(* CoDeSys 2.3.9.41 project: KS Griazovetskaya(ver27.07.20, manStopN0204).pro *)
(* Libraries: PID_Regulators.lib 6.11.19 15:29:27, Util.lib 18.5.10 15:14:28, STANDARD.LIB 4.10.05 11:14:46, IECSFC.LIB 13.4.06 15:51:28, ANALYZATION.LIB 5.10.99 09:05:06 *)

(* PLC configuration (modules and I/O channels)
Fast discrete inputs [I_SIMPLE_INPUT] node 0, in %IB0 out %QB0 {Filtrationtime = 10}
  DD1_DI0 AT %IX0.0 [BitInput] резерв
  DD1_DI1 AT %IX0.1 [BitInput] резерв
  DD1_DI2 AT %IX0.2 [BitInput] резерв
  DD1_DI3 AT %IX0.3 [BitInput] резерв
Discrete inputs [ID130] node 1, in %IB1 out %QB1 {Filtrationtime_GeneralINP = 10; Visibility = No; PinCount = 12}
  AT %IB1.0 [ByteInput] 8 discrete inputs
  AT %IB1.1 [ByteInput] 4 discrete inputs
Discrete outputs [ID131] node 2, in %IB2 out %QB2 {SafeValueByte = 0; SafeValueByteM = 0; Visibility = No; PinCount = 12}
  AT %QB2.0 [ByteOutput] 8 discrete outputs
  AT %QB2.1 [ByteOutput] 4 discrete outputs
Fast analog inputs [ID125] node 3, in %IB3 out %QB3 {Flt_Comm = 50Hz 2Por}
  DD1_AI0 AT %IR3.0 [FloatInputP] AI #1 - датчик температуры в помещении (метран) {AIN_TYPE = 4-20 mA; Peak_Filtr = 200; Flt_Ch = Off; TauRC = 10; MinFV = 0; MaxFV = 100}
  DD1_AI1 AT %IR3.1 [FloatInputP] AI #2 - расходомер FT01.01 (на входе, до отстойника) {AIN_TYPE = 4-20 mA; Peak_Filtr = 200; Flt_Ch = Off; TauRC = 10; MinFV = 0; MaxFV = 600}
  DD1_AI2 AT %IR3.2 [FloatInputP] AI #3 - расходомер FT01.02 (на выходе, после отстойника) {AIN_TYPE = 4-20 mA; Peak_Filtr = 200; Flt_Ch = Off; TauRC = 10; MinFV = 0; MaxFV = 600}
  DD1_AI3 AT %IR3.3 [FloatInputP] AI #4 - рН-метр QE01.01 (на входе, до отстойника) {AIN_TYPE = 4-20 mA; Peak_Filtr = 200; Flt_Ch = Off; TauRC = 10; MinFV = 0; MaxFV = 14}
  DD1_AI4 AT %IR3.4 [FloatInputP] AI #5 - рН-метр QE01.02 (на выходе, после отстойника) {AIN_TYPE = 4-20 mA; Peak_Filtr = 200; Flt_Ch = Off; TauRC = 10; MinFV = 0; MaxFV = 14}
  DD1_AI5 AT %IR3.5 [FloatInputP] AI #6 - сигнал от ФПК, давление на входе {AIN_TYPE = 4-20 mA; Peak_Filtr = 200; Flt_Ch = Off; TauRC = 10; MinFV = 0; MaxFV = 16}
  DD1_AI6 AT %IR3.6 [FloatInputP] AI #7 - резерв {AIN_TYPE = 4-20 mA; Peak_Filtr = 200; Flt_Ch = Off; TauRC = 10; MinFV = 0; MaxFV = 20000.0}
  DD1_AI7 AT %IR3.7 [FloatInputP] AI#8 - резерв {AIN_TYPE = 4-20 mA; Peak_Filtr = 200; Flt_Ch = Off; TauRC = 10; MinFV = 0; MaxFV = 20000.0}
  AT %IW3.8 [WordInput] AI read time (10ms)
Analog outputs [ID126] node 4, in %IB4 out %QB4
  DD1_AO0 AT %QR4.0 [FloatOutputP] AO #1 - управление ЧРП Н01.05 (поддержание расхода по расходомеру FT01.02) {AOUT_TYPE = 4-20 mA; SafeValueREAL = 0.0}
  DD1_AO1 AT %QR4.1 [FloatOutputP] AO #2 - управление ЧРП НД08.03/01 (подача флокулянта на входе, до отстойника, по FT01.01) {AOUT_TYPE = 4-20 mA; SafeValueREAL = 0.0}
  DD1_AO2 AT %QR4.2 [FloatOutputP] AO #3 - управление ЧРП НД08.03/02 (подача флокулянта на входе, до отстойника, по FT01.01) {AOUT_TYPE = 4-20 mA; SafeValueREAL = 0.0}
  DD1_AO3 AT %QR4.3 [FloatOutputP] AO #4 - управление НД05.02/01 (подача 10%NaCl из УПГ на входе, до отстойника, по FT01.01) {AOUT_TYPE = 4-20 mA; SafeValueREAL = 0.0}
Special input [ID103] node 5, in %IB5 out %QB5 {Filtrationtime = 1000; PinCount = 1; WatchDogPeriod = 400; PollPeriod = 3000; Visibility = No}
  AT %IX5.0 [BitInput] Special input
Special output [ID104] node 6, in %IB6 out %QB6 {Visibility = No; PinCount = 1}
  AT %QX6.0 [BitOutput] Special output
ModBus (Master) [MODBUS_MASTER_ID450] node 7, in %IB7 out %QB7 {Visibility = No}
  lastAddress AT %QD7.0 [DWordOutput] Last address
  lastError AT %QW7.1 [WordOutput] Last error
  RS-485-1 [COM1_USART] node 0, in %IB7.0 out %QB7.0 {CommunicationSpeed = 9600; Parity = EVEN; BitLength = 8 bits; StopLength = One stop bit; InterfaceType = RS485; FrameOriented = RTU; Timeout = 0; Visibility = No}
  Universal Modbus device [ID2000] node 1, in %IB7.1 out %QB7.1 {ModuleIP = 10:0:0:102; ServiceTimeout = 20; TCPport = 502; NetMode = Serial; ModuleSlaveAddress = 2; RequestType = Both; PeriodOfService = 100; Visibility = No; RepeatCounter = 0; ByteSequence = Trace_mode}
    AT %QB7.1.0 [ComChannel] Command (0xff - Start)
DD2_DO AT %QD7.1.0.0 [DWordOutput] регистр 0, команда 0х0f
Universal Modbus device [ID2000] node 2, in %IB7.2 out %QB7.2 {ModuleIP = 10:0:0:103; ServiceTimeout = 20; TCPport = 502; NetMode = Serial; ModuleSlaveAddress = 3; RequestType = Both; PeriodOfService = 100; Visibility = No; RepeatCounter = 0; ByteSequence = Trace_mode}
  AT %QB7.2.0 [ComChannel] Command (0xff - Start)
DD3_DO AT %QD7.2.0.0 [DWordOutput]
Universal Modbus device [ID2000] node 3, in %IB7.3 out %QB7.3 {ModuleIP = 10:0:0:104; ServiceTimeout = 20; TCPport = 502; NetMode = Serial; ModuleSlaveAddress = 4; RequestType = Both; PeriodOfService = 100; Visibility = No; RepeatCounter = 0; ByteSequence = Trace_mode}
  AT %QB7.3.0 [ComChannel] Command (0xff - Start)
  32bit output module [ID2006] node 0, in %IB7.3.0 out %QB7.3.0 {ModbusAddress = 0; Command_write_regs = Force multiple coils (0x0f); Visibility = No}
    DD4_DO AT %QD7.3.0.0 [DWordOutput]
Universal Modbus device [ID2000] node 4, in %IB7.4 out %QB7.4 {ModuleIP = 10:0:0:105; ServiceTimeout = 20; TCPport = 502; NetMode = Serial; ModuleSlaveAddress = 5; RequestType = Both; PeriodOfService = 100; Visibility = No; RepeatCounter = 0; ByteSequence = Trace_mode}
  AT %QB7.4.0 [ComChannel] Command (0xff - Start)
DD5_DI AT %ID7.4.0.0 [DWordInput]
Universal Modbus device [ID2000] node 5, in %IB7.5 out %QB7.5 {ModuleIP = 10:0:0:106; ServiceTimeout = 20; TCPport = 502; NetMode = Serial; ModuleSlaveAddress = 6; RequestType = Both; PeriodOfService = 100; Visibility = No; RepeatCounter = 0; ByteSequence = Trace_mode}
  AT %QB7.5.0 [ComChannel] Command (0xff - Start)
DD6_DI AT %ID7.5.0.0 [DWordInput]
Universal Modbus device [ID2000] node 6, in %IB7.6 out %QB7.6 {ModuleIP = 10:0:0:107; ServiceTimeout = 20; TCPport = 502; NetMode = Serial; ModuleSlaveAddress = 7; RequestType = Both; PeriodOfService = 100; Visibility = No; RepeatCounter = 0; ByteSequence = Trace_mode}
  AT %QB7.6.0 [ComChannel] Command (0xff - Start)
DD7_DI AT %ID7.6.0.0 [DWordInput]
Universal Modbus device [ID2000] node 7, in %IB7.7 out %QB7.7 {ModuleIP = 10:0:0:108; ServiceTimeout = 20; TCPport = 502; NetMode = Serial; ModuleSlaveAddress = 8; RequestType = Both; PeriodOfService = 100; Visibility = No; RepeatCounter = 0; ByteSequence = Trace_mode}
  AT %QB7.7.0 [ComChannel] Command (0xff - Start)
DD8_DI AT %ID7.7.0.0 [DWordInput]
Universal Modbus device [ID2000] node 8, in %IB7.8 out %QB7.8 {ModuleIP = 10:0:0:109; ServiceTimeout = 20; TCPport = 502; NetMode = Serial; ModuleSlaveAddress = 9; RequestType = Both; PeriodOfService = 100; Visibility = No; RepeatCounter = 0; ByteSequence = Trace_mode}
  AT %QB7.8.0 [ComChannel] Command (0xff - Start)
DD9_DI AT %ID7.8.0.0 [DWordInput]
Universal Modbus device [ID2000] node 9, in %IB7.9 out %QB7.9 {ModuleIP = 10:0:0:110; ServiceTimeout = 20; TCPport = 502; NetMode = Serial; ModuleSlaveAddress = 10; RequestType = Both; PeriodOfService = 100; Visibility = No; RepeatCounter = 0; ByteSequence = Trace_mode}
  AT %QB7.9.0 [ComChannel] Command (0xff - Start)
DD10_AO0 AT %QW7.9.0.0 [WordOutput] управление 4...20мА НД05.02/02
DD10_AO1 AT %QW7.9.1.0 [WordOutput] управление 4...20мА НД06.02/01
DD10_AO2 AT %QW7.9.2.0 [WordOutput] управление 4...20мА НД06.02/02
DD10_AO3 AT %QW7.9.3.0 [WordOutput] управление 4...20мА НД06.03/01
DD10_AO4 AT %QW7.9.4.0 [WordOutput] управление 4...20мА НД06.03/02
DD10_AO5 AT %QW7.9.5.0 [WordOutput] управление 4...20мА НД07.03/01
DD10_AO6 AT %QW7.9.6.0 [WordOutput] управление 4...20мА НД07.03/02
DD10_AO7 AT %QW7.9.7.0 [WordOutput] управление 4...20мА НД08.04
Universal Modbus device [ID2000] node 10, in %IB7.10 out %QB7.10 {ModuleIP = 10:0:0:223; ServiceTimeout = 20; TCPport = 502; NetMode = Serial; ModuleSlaveAddress = 11; RequestType = By value change; PeriodOfService = 100; Visibility = No; RepeatCounter = 0; ByteSequence = Trace_mode}
  AT %QB7.10.0 [ComChannel] Command (0xff - Start)
AT %QB7.10.0.0 [ByteOutput]
Universal Modbus device [ID2000] node 11, in %IB7.11 out %QB7.11 {ModuleIP = 10:0:0:223; ServiceTimeout = 20; TCPport = 502; NetMode = Serial; ModuleSlaveAddress = 11; RequestType = By poll time; PeriodOfService = 100; Visibility = No; RepeatCounter = 0; ByteSequence = Trace_mode}
  AT %QB7.11.0 [ComChannel] Command (0xff - Start)
AT %IB7.11.0.0 [ByteInput]
Universal Modbus device [ID2000] node 12, in %IB7.12 out %QB7.12 {ModuleIP = 10:0:0:223; ServiceTimeout = 20; TCPport = 502; NetMode = Serial; ModuleSlaveAddress = 12; RequestType = By value change; PeriodOfService = 100; Visibility = No; RepeatCounter = 0; ByteSequence = Trace_mode}
  AT %QB7.12.0 [ComChannel] Command (0xff - Start)
AT %QB7.12.0.0 [ByteOutput]
Universal Modbus device [ID2000] node 13, in %IB7.13 out %QB7.13 {ModuleIP = 10:0:0:223; ServiceTimeout = 20; TCPport = 502; NetMode = Serial; ModuleSlaveAddress = 12; RequestType = By poll time; PeriodOfService = 100; Visibility = No; RepeatCounter = 0; ByteSequence = Trace_mode}
  AT %QB7.13.0 [ComChannel] Command (0xff - Start)
AT %IB7.13.0.0 [ByteInput]
AT %QD8.0 [DWordOutput] Last address
AT %QW8.1 [WordOutput] Last error
RS-232 [COM2_USART] node 0, in %IB8.0 out %QB8.0 {CommunicationSpeed = 57600; Parity = NO PARITY CHECK; BitLength = 8 bits; StopLength = One stop bit; InterfaceType = RS232; FrameOriented = RTU; Timeout = 0; Visibility = No}
Universal Modbus device [ID2000] node 1, in %IB8.1 out %QB8.1 {ModuleIP = 10:0:0:223; ServiceTimeout = 150; TCPport = 502; NetMode = Serial; ModuleSlaveAddress = 1; RequestType = By value change; PeriodOfService = 100; Visibility = No; RepeatCounter = 0; ByteSequence = Native}
  AT %QB8.1.0 [ComChannel] Command (0xff - Start)
  Real output module [ID2008] node 0, in %IB8.1.0 out %QB8.1.0 {ModbusAddress = 256; Command_write_regs = Preset multiple Registers (0x10); Visibility = No}
    panFT0101value AT %QD8.1.0.0 [FloatOutput]
  Real output module [ID2008] node 1, in %IB8.1.1 out %QB8.1.1 {ModbusAddress = 258; Command_write_regs = Preset multiple Registers (0x10); Visibility = No}
    panQE0101value AT %QD8.1.1.0 [FloatOutput]
  Real output module [ID2008] node 2, in %IB8.1.2 out %QB8.1.2 {ModbusAddress = 260; Command_write_regs = Preset multiple Registers (0x10); Visibility = No}
    panFT0102value AT %QD8.1.2.0 [FloatOutput]
  Real output module [ID2008] node 3, in %IB8.1.3 out %QB8.1.3 {ModbusAddress = 262; Command_write_regs = Preset multiple Registers (0x10); Visibility = No}
    panQE0102value AT %QD8.1.3.0 [FloatOutput]
  Real output module [ID2008] node 4, in %IB8.1.4 out %QB8.1.4 {ModbusAddress = 264; Command_write_regs = Preset multiple Registers (0x10); Visibility = No}
    panFPKpressureValue AT %QD8.1.4.0 [FloatOutput]
  Real output module [ID2008] node 5, in %IB8.1.5 out %QB8.1.5 {ModbusAddress = 266; Command_write_regs = Preset multiple Registers (0x10); Visibility = No}
    panFQS0301total AT %QD8.1.5.0 [FloatOutput]
  Real output module [ID2008] node 6, in %IB8.1.6 out %QB8.1.6 {ModbusAddress = 268; Command_write_regs = Preset multiple Registers (0x10); Visibility = No}
    panTemperature AT %QD8.1.6.0 [FloatOutput]
  Register output module [ID2004] node 7, in %IB8.1.7 out %QB8.1.7 {ModbusAddress = 270; Command_write_one_reg = Write multiple registers(0x10); Visibility = No}
    panND050201workDays AT %QW8.1.7.0 [WordOutput]
  Register output module [ID2004] node 8, in %IB8.1.8 out %QB8.1.8 {ModbusAddress = 271; Command_write_one_reg = Write multiple registers(0x10); Visibility = No}
    panND050201workHours AT %QW8.1.8.0 [WordOutput]
  Register output module [ID2004] node 9, in %IB8.1.9 out %QB8.1.9 {ModbusAddress = 272; Command_write_one_reg = Write multiple registers(0x10); Visibility = No}
    panND050201workMinutes AT %QW8.1.9.0 [WordOutput]
  Register output module [ID2004] node 10, in %IB8.1.10 out %QB8.1.10 {ModbusAddress = 273; Command_write_one_reg = Write multiple registers(0x10); Visibility = No}
    panND050201workSeconds AT %QW8.1.10.0 [WordOutput]
  Register output module [ID2004] node 11, in %IB8.1.11 out %QB8.1.11 {ModbusAddress = 274; Command_write_one_reg = Write multiple registers(0x10); Visibility = No}
    panND050202workDays AT %QW8.1.11.0 [WordOutput]
  Register output module [ID2004] node 12, in %IB8.1.12 out %QB8.1.12 {ModbusAddress = 275; Command_write_one_reg = Write multiple registers(0x10); Visibility = No}
    panND050202workHours AT %QW8.1.12.0 [WordOutput]
  Register output module [ID2004] node 13, in %IB8.1.13 out %QB8.1.13 {ModbusAddress = 276; Command_write_one_reg = Write multiple registers(0x10); Visibility = No}
    panND050202workMinutes AT %QW8.1.13.0 [WordOutput]
  Register output module [ID2004] node 14, in %IB8.1.14 out %QB8.1.14 {ModbusAddress = 277; Command_write_one_reg = Write multiple registers(0x10); Visibility = No}
    panND050202workSeconds AT %QW8.1.14.0 [WordOutput]
  Register output module [ID2004] node 15, in %IB8.1.15 out %QB8.1.15 {ModbusAddress = 278; Command_write_one_reg = Write multiple registers(0x10); Visibility = No}
    panND0502counterP1 AT %QW8.1.15.0 [WordOutput]
  Register output module [ID2004] node 16, in %IB8.1.16 out %QB8.1.16 {ModbusAddress = 279; Command_write_one_reg = Write multiple registers(0x10); Visibility = No}
    panND0502counterP2 AT %QW8.1.16.0 [WordOutput]
  Register output module [ID2004] node 17, in %IB8.1.17 out %QB8.1.17 {ModbusAddress = 280; Command_write_one_reg = Write multiple registers(0x10); Visibility = No}
    panND060201workDays AT %QW8.1.17.0 [WordOutput]
  Register output module [ID2004] node 18, in %IB8.1.18 out %QB8.1.18 {ModbusAddress = 281; Command_write_one_reg = Write multiple registers(0x10); Visibility = No}
    panND060201workHours AT %QW8.1.18.0 [WordOutput]
  Register output module [ID2004] node 19, in %IB8.1.19 out %QB8.1.19 {ModbusAddress = 282; Command_write_one_reg = Write multiple registers(0x10); Visibility = No}
    panND060201workMinutes AT %QW8.1.19.0 [WordOutput]
  Register output module [ID2004] node 20, in %IB8.1.20 out %QB8.1.20 {ModbusAddress = 283; Command_write_one_reg = Write multiple registers(0x10); Visibility = No}
    panND060201workSeconds AT %QW8.1.20.0 [WordOutput]
  Register output module [ID2004] node 21, in %IB8.1.21 out %QB8.1.21 {ModbusAddress = 284; Command_write_one_reg = Write multiple registers(0x10); Visibility = No}
    panND060202workDays AT %QW8.1.21.0 [WordOutput]
  Register output module [ID2004] node 22, in %IB8.1.22 out %QB8.1.22 {ModbusAddress = 285; Command_write_one_reg = Write multiple registers(0x10); Visibility = No}
    panND060202workHours AT %QW8.1.22.0 [WordOutput]
  Register output module [ID2004] node 23, in %IB8.1.23 out %QB8.1.23 {ModbusAddress = 286; Command_write_one_reg = Write multiple registers(0x10); Visibility = No}
    panND060202workMinutes AT %QW8.1.23.0 [WordOutput]
  Register output module [ID2004] node 24, in %IB8.1.24 out %QB8.1.24 {ModbusAddress = 287; Command_write_one_reg = Write multiple registers(0x10); Visibility = No}
    panND060202workSeconds AT %QW8.1.24.0 [WordOutput]
  Register output module [ID2004] node 25, in %IB8.1.25 out %QB8.1.25 {ModbusAddress = 288; Command_write_one_reg = Write multiple registers(0x10); Visibility = No}
    panND0602counterP1 AT %QW8.1.25.0 [WordOutput]
  Register output module [ID2004] node 26, in %IB8.1.26 out %QB8.1.26 {ModbusAddress = 289; Command_write_one_reg = Write multiple registers(0x10); Visibility = No}
    panND0602counterP2 AT %QW8.1.26.0 [WordOutput]
  Register output module [ID2004] node 27, in %IB8.1.27 out %QB8.1.27 {ModbusAddress = 290; Command_write_one_reg = Write multiple registers(0x10); Visibility = No}
    panND060301workDays AT %QW8.1.27.0 [WordOutput]
  Register output module [ID2004] node 28, in %IB8.1.28 out %QB8.1.28 {ModbusAddress = 291; Command_write_one_reg = Write multiple registers(0x10); Visibility = No}
    panND060301workHours AT %QW8.1.28.0 [WordOutput]
  Register output module [ID2004] node 29, in %IB8.1.29 out %QB8.1.29 {ModbusAddress = 292; Command_write_one_reg = Write multiple registers(0x10); Visibility = No}
    panND060301workMinutes AT %QW8.1.29.0 [WordOutput]
  Register output module [ID2004] node 30, in %IB8.1.30 out %QB8.1.30 {ModbusAddress = 293; Command_write_one_reg = Write multiple registers(0x10); Visibility = No}
    panND060301workSeconds AT %QW8.1.30.0 [WordOutput]
  Register output module [ID2004] node 31, in %IB8.1.31 out %QB8.1.31 {ModbusAddress = 294; Command_write_one_reg = Write multiple registers(0x10); Visibility = No}
    panND060302workDays AT %QW8.1.31.0 [WordOutput]
  Register output module [ID2004] node 32, in %IB8.1.32 out %QB8.1.32 {ModbusAddress = 295; Command_write_one_reg = Write multiple registers(0x10); Visibility = No}
    panND060302workHours AT %QW8.1.32.0 [WordOutput]
  Register output module [ID2004] node 33, in %IB8.1.33 out %QB8.1.33 {ModbusAddress = 296; Command_write_one_reg = Write multiple registers(0x10); Visibility = No}
    panND060302workMinutes AT %QW8.1.33.0 [WordOutput]
  Register output module [ID2004] node 34, in %IB8.1.34 out %QB8.1.34 {ModbusAddress = 297; Command_write_one_reg = Write multiple registers(0x10); Visibility = No}
    panND060302workSeconds AT %QW8.1.34.0 [WordOutput]
  Register output module [ID2004] node 35, in %IB8.1.35 out %QB8.1.35 {ModbusAddress = 298; Command_write_one_reg = Write multiple registers(0x10); Visibility = No}
    panND0603counterP1 AT %QW8.1.35.0 [WordOutput]
  Register output module [ID2004] node 36, in %IB8.1.36 out %QB8.1.36 {ModbusAddress = 299; Command_write_one_reg = Write multiple registers(0x10); Visibility = No}
    panND0603counterP2 AT %QW8.1.36.0 [WordOutput]
  Register output module [ID2004] node 37, in %IB8.1.37 out %QB8.1.37 {ModbusAddress = 300; Command_write_one_reg = Write multiple registers(0x10); Visibility = No}
    panND070301workDays AT %QW8.1.37.0 [WordOutput]
  Register output module [ID2004] node 38, in %IB8.1.38 out %QB8.1.38 {ModbusAddress = 301; Command_write_one_reg = Write multiple registers(0x10); Visibility = No}
    panND070301workHours AT %QW8.1.38.0 [WordOutput]
  Register output module [ID2004] node 39, in %IB8.1.39 out %QB8.1.39 {ModbusAddress = 302; Command_write_one_reg = Write multiple registers(0x10); Visibility = No}
    panND070301workMinutes AT %QW8.1.39.0 [WordOutput]
  Register output module [ID2004] node 40, in %IB8.1.40 out %QB8.1.40 {ModbusAddress = 303; Command_write_one_reg = Write multiple registers(0x10); Visibility = No}
    panND070301workSeconds AT %QW8.1.40.0 [WordOutput]
  Register output module [ID2004] node 41, in %IB8.1.41 out %QB8.1.41 {ModbusAddress = 304; Command_write_one_reg = Write multiple registers(0x10); Visibility = No}
    panND070302workDays AT %QW8.1.41.0 [WordOutput]
  Register output module [ID2004] node 42, in %IB8.1.42 out %QB8.1.42 {ModbusAddress = 305; Command_write_one_reg = Write multiple registers(0x10); Visibility = No}
    panND070302workHours AT %QW8.1.42.0 [WordOutput]
  Register output module [ID2004] node 43, in %IB8.1.43 out %QB8.1.43 {ModbusAddress = 306; Command_write_one_reg = Write multiple registers(0x10); Visibility = No}
    panND070302workMinutes AT %QW8.1.43.0 [WordOutput]
  Register output module [ID2004] node 44, in %IB8.1.44 out %QB8.1.44 {ModbusAddress = 307; Command_write_one_reg = Write multiple registers(0x10); Visibility = No}
    panND070302workSeconds AT %QW8.1.44.0 [WordOutput]
  Register output module [ID2004] node 45, in %IB8.1.45 out %QB8.1.45 {ModbusAddress = 308; Command_write_one_reg = Write multiple registers(0x10); Visibility = No}
    panND0703counterP1 AT %QW8.1.45.0 [WordOutput]
  Register output module [ID2004] node 46, in %IB8.1.46 out %QB8.1.46 {ModbusAddress = 309; Command_write_one_reg = Write multiple registers(0x10); Visibility = No}
    panND0703counterP2 AT %QW8.1.46.0 [WordOutput]
  Register output module [ID2004] node 47, in %IB8.1.47 out %QB8.1.47 {ModbusAddress = 310; Command_write_one_reg = Write multiple registers(0x10); Visibility = No}
    panND080301workDays AT %QW8.1.47.0 [WordOutput]
  Register output module [ID2004] node 48, in %IB8.1.48 out %QB8.1.48 {ModbusAddress = 311; Command_write_one_reg = Write multiple registers(0x10); Visibility = No}
    panND080301workHours AT %QW8.1.48.0 [WordOutput]
  Register output module [ID2004] node 49, in %IB8.1.49 out %QB8.1.49 {ModbusAddress = 312; Command_write_one_reg = Write multiple registers(0x10); Visibility = No}
    panND080301workMinutes AT %QW8.1.49.0 [WordOutput]
  Register output module [ID2004] node 50, in %IB8.1.50 out %QB8.1.50 {ModbusAddress = 313; Command_write_one_reg = Write multiple registers(0x10); Visibility = No}
    panND080301workSeconds AT %QW8.1.50.0 [WordOutput]
  Register output module [ID2004] node 51, in %IB8.1.51 out %QB8.1.51 {ModbusAddress = 314; Command_write_one_reg = Write multiple registers(0x10); Visibility = No}
    panND080302workDays AT %QW8.1.51.0 [WordOutput]
  Register output module [ID2004] node 52, in %IB8.1.52 out %QB8.1.52 {ModbusAddress = 315; Command_write_one_reg = Write multiple registers(0x10); Visibility = No}
    panND080302workHours AT %QW8.1.52.0 [WordOutput]
  Register output module [ID2004] node 53, in %IB8.1.53 out %QB8.1.53 {ModbusAddress = 316; Command_write_one_reg = Write multiple registers(0x10); Visibility = No}
    panND080302workMinutes AT %QW8.1.53.0 [WordOutput]
  Register output module [ID2004] node 54, in %IB8.1.54 out %QB8.1.54 {ModbusAddress = 317; Command_write_one_reg = Write multiple registers(0x10); Visibility = No}
    panND080302workSeconds AT %QW8.1.54.0 [WordOutput]
  Register output module [ID2004] node 55, in %IB8.1.55 out %QB8.1.55 {ModbusAddress = 318; Command_write_one_reg = Write multiple registers(0x10); Visibility = No}
    panND0803counterP1 AT %QW8.1.55.0 [WordOutput]
  Register output module [ID2004] node 56, in %IB8.1.56 out %QB8.1.56 {ModbusAddress = 319; Command_write_one_reg = Write multiple registers(0x10); Visibility = No}
    panND0803counterP2 AT %QW8.1.56.0 [WordOutput]
  Register output module [ID2004] node 57, in %IB8.1.57 out %QB8.1.57 {ModbusAddress = 320; Command_write_one_reg = Write multiple registers(0x10); Visibility = No}
    panN010501workDays AT %QW8.1.57.0 [WordOutput]
  Register output module [ID2004] node 58, in %IB8.1.58 out %QB8.1.58 {ModbusAddress = 321; Command_write_one_reg = Write multiple registers(0x10); Visibility = No}
    panN010501workHours AT %QW8.1.58.0 [WordOutput]
  Register output module [ID2004] node 59, in %IB8.1.59 out %QB8.1.59 {ModbusAddress = 322; Command_write_one_reg = Write multiple registers(0x10); Visibility = No}
    panN010501workMinutes AT %QW8.1.59.0 [WordOutput]
  Register output module [ID2004] node 60, in %IB8.1.60 out %QB8.1.60 {ModbusAddress = 323; Command_write_one_reg = Write multiple registers(0x10); Visibility = No}
    panN010501workSeconds AT %QW8.1.60.0 [WordOutput]
  Register output module [ID2004] node 61, in %IB8.1.61 out %QB8.1.61 {ModbusAddress = 324; Command_write_one_reg = Write multiple registers(0x10); Visibility = No}
    panN010502workDays AT %QW8.1.61.0 [WordOutput]
  Register output module [ID2004] node 62, in %IB8.1.62 out %QB8.1.62 {ModbusAddress = 325; Command_write_one_reg = Write multiple registers(0x10); Visibility = No}
    panN010502workHours AT %QW8.1.62.0 [WordOutput]
  Register output module [ID2004] node 63, in %IB8.1.63 out %QB8.1.63 {ModbusAddress = 326; Command_write_one_reg = Write multiple registers(0x10); Visibility = No}
    panN010502workMinutes AT %QW8.1.63.0 [WordOutput]
  Register output module [ID2004] node 64, in %IB8.1.64 out %QB8.1.64 {ModbusAddress = 327; Command_write_one_reg = Write multiple registers(0x10); Visibility = No}
    panN010502workSeconds AT %QW8.1.64.0 [WordOutput]
  Register output module [ID2004] node 65, in %IB8.1.65 out %QB8.1.65 {ModbusAddress = 328; Command_write_one_reg = Write multiple registers(0x10); Visibility = No}
    panN0105counterP1 AT %QW8.1.65.0 [WordOutput]
  Register output module [ID2004] node 66, in %IB8.1.66 out %QB8.1.66 {ModbusAddress = 329; Command_write_one_reg = Write multiple registers(0x10); Visibility = No}
    panN0105counterP2 AT %QW8.1.66.0 [WordOutput]
  Register output module [ID2004] node 67, in %IB8.1.67 out %QB8.1.67 {ModbusAddress = 330; Command_write_one_reg = Write multiple registers(0x10); Visibility = No}
    panN020401workDays AT %QW8.1.67.0 [WordOutput]
  Register output module [ID2004] node 68, in %IB8.1.68 out %QB8.1.68 {ModbusAddress = 331; Command_write_one_reg = Write multiple registers(0x10); Visibility = No}
    panN020401workHours AT %QW8.1.68.0 [WordOutput]
  Register output module [ID2004] node 69, in %IB8.1.69 out %QB8.1.69 {ModbusAddress = 332; Command_write_one_reg = Write multiple registers(0x10); Visibility = No}
    panN020401workMinutes AT %QW8.1.69.0 [WordOutput]
  Register output module [ID2004] node 70, in %IB8.1.70 out %QB8.1.70 {ModbusAddress = 333; Command_write_one_reg = Write multiple registers(0x10); Visibility = No}
    panN020401workSeconds AT %QW8.1.70.0 [WordOutput]
  Register output module [ID2004] node 71, in %IB8.1.71 out %QB8.1.71 {ModbusAddress = 334; Command_write_one_reg = Write multiple registers(0x10); Visibility = No}
    panN020402workDays AT %QW8.1.71.0 [WordOutput]
  Register output module [ID2004] node 72, in %IB8.1.72 out %QB8.1.72 {ModbusAddress = 335; Command_write_one_reg = Write multiple registers(0x10); Visibility = No}
    panN020402workHours AT %QW8.1.72.0 [WordOutput]
  Register output module [ID2004] node 73, in %IB8.1.73 out %QB8.1.73 {ModbusAddress = 336; Command_write_one_reg = Write multiple registers(0x10); Visibility = No}
    panN020402workMinutes AT %QW8.1.73.0 [WordOutput]
  Register output module [ID2004] node 74, in %IB8.1.74 out %QB8.1.74 {ModbusAddress = 337; Command_write_one_reg = Write multiple registers(0x10); Visibility = No}
    panN020402workSeconds AT %QW8.1.74.0 [WordOutput]
  Register output module [ID2004] node 75, in %IB8.1.75 out %QB8.1.75 {ModbusAddress = 338; Command_write_one_reg = Write multiple registers(0x10); Visibility = No}
    panN0204counterP1 AT %QW8.1.75.0 [WordOutput]
  Register output module [ID2004] node 76, in %IB8.1.76 out %QB8.1.76 {ModbusAddress = 339; Command_write_one_reg = Write multiple registers(0x10); Visibility = No}
    panN0204counterP2 AT %QW8.1.76.0 [WordOutput]
  Register output module [ID2004] node 77, in %IB8.1.77 out %QB8.1.77 {ModbusAddress = 340; Command_write_one_reg = Write multiple registers(0x10); Visibility = No}
    panN040401workDays AT %QW8.1.77.0 [WordOutput]
  Register output module [ID2004] node 78, in %IB8.1.78 out %QB8.1.78 {ModbusAddress = 341; Command_write_one_reg = Write multiple registers(0x10); Visibility = No}
    panN040401workHours AT %QW8.1.78.0 [WordOutput]
  Register output module [ID2004] node 79, in %IB8.1.79 out %QB8.1.79 {ModbusAddress = 342; Command_write_one_reg = Write multiple registers(0x10); Visibility = No}
    panN040401workMinutes AT %QW8.1.79.0 [WordOutput]
  Register output module [ID2004] node 80, in %IB8.1.80 out %QB8.1.80 {ModbusAddress = 343; Command_write_one_reg = Write multiple registers(0x10); Visibility = No}
    panN040401workSeconds AT %QW8.1.80.0 [WordOutput]
  Register output module [ID2004] node 81, in %IB8.1.81 out %QB8.1.81 {ModbusAddress = 344; Command_write_one_reg = Write multiple registers(0x10); Visibility = No}
    panN040402workDays AT %QW8.1.81.0 [WordOutput]
  Register output module [ID2004] node 82, in %IB8.1.82 out %QB8.1.82 {ModbusAddress = 345; Command_write_one_reg = Write multiple registers(0x10); Visibility = No}
    panN040402workHours AT %QW8.1.82.0 [WordOutput]
  Register output module [ID2004] node 83, in %IB8.1.83 out %QB8.1.83 {ModbusAddress = 346; Command_write_one_reg = Write multiple registers(0x10); Visibility = No}
    panN040402workMinutes AT %QW8.1.83.0 [WordOutput]
  Register output module [ID2004] node 84, in %IB8.1.84 out %QB8.1.84 {ModbusAddress = 347; Command_write_one_reg = Write multiple registers(0x10); Visibility = No}
    panN040402workSeconds AT %QW8.1.84.0 [WordOutput]
  Register output module [ID2004] node 85, in %IB8.1.85 out %QB8.1.85 {ModbusAddress = 348; Command_write_one_reg = Write multiple registers(0x10); Visibility = No}
    panN0404counterP1 AT %QW8.1.85.0 [WordOutput]
  Register output module [ID2004] node 86, in %IB8.1.86 out %QB8.1.86 {ModbusAddress = 349; Command_write_one_reg = Write multiple registers(0x10); Visibility = No}
    panN0404counterP2 AT %QW8.1.86.0 [WordOutput]
  Register output module [ID2004] node 87, in %IB8.1.87 out %QB8.1.87 {ModbusAddress = 350; Command_write_one_reg = Write multiple registers(0x10); Visibility = No}
    panUFO030101workDays AT %QW8.1.87.0 [WordOutput]
  Register output module [ID2004] node 88, in %IB8.1.88 out %QB8.1.88 {ModbusAddress = 351; Command_write_one_reg = Write multiple registers(0x10); Visibility = No}
    panUFO030101workHours AT %QW8.1.88.0 [WordOutput]
  Register output module [ID2004] node 89, in %IB8.1.89 out %QB8.1.89 {ModbusAddress = 352; Command_write_one_reg = Write multiple registers(0x10); Visibility = No}
    panUFO030101workMinutes AT %QW8.1.89.0 [WordOutput]
  Register output module [ID2004] node 90, in %IB8.1.90 out %QB8.1.90 {ModbusAddress = 353; Command_write_one_reg = Write multiple registers(0x10); Visibility = No}
    panUFO030101workSeconds AT %QW8.1.90.0 [WordOutput]
  Register output module [ID2004] node 91, in %IB8.1.91 out %QB8.1.91 {ModbusAddress = 354; Command_write_one_reg = Write multiple registers(0x10); Visibility = No}
    panUFO030102workDays AT %QW8.1.91.0 [WordOutput]
  Register output module [ID2004] node 92, in %IB8.1.92 out %QB8.1.92 {ModbusAddress = 355; Command_write_one_reg = Write multiple registers(0x10); Visibility = No}
    panUFO030102workHours AT %QW8.1.92.0 [WordOutput]
  Register output module [ID2004] node 93, in %IB8.1.93 out %QB8.1.93 {ModbusAddress = 356; Command_write_one_reg = Write multiple registers(0x10); Visibility = No}
    panUFO030102workMinutes AT %QW8.1.93.0 [WordOutput]
  Register output module [ID2004] node 94, in %IB8.1.94 out %QB8.1.94 {ModbusAddress = 357; Command_write_one_reg = Write multiple registers(0x10); Visibility = No}
    panUFO030102workSeconds AT %QW8.1.94.0 [WordOutput]
  Register output module [ID2004] node 95, in %IB8.1.95 out %QB8.1.95 {ModbusAddress = 358; Command_write_one_reg = Write multiple registers(0x10); Visibility = No}
    panUFO0301counterP1 AT %QW8.1.95.0 [WordOutput]
  Register output module [ID2004] node 96, in %IB8.1.96 out %QB8.1.96 {ModbusAddress = 359; Command_write_one_reg = Write multiple registers(0x10); Visibility = No}
    panUFO0301counterP2 AT %QW8.1.96.0 [WordOutput]
panVolumeToRegen AT %QD8.1.97.0 [FloatOutput]
8 bit output module [ID2002] node 98, in %IB8.1.98 out %QB8.1.98 {ModbusAddress = 256; Command_write_byte = Force multiply coils (0x0f); Visibility = No}
  AT %QB8.1.98.0 [ByteOutput]
8 bit output module [ID2002] node 99, in %IB8.1.99 out %QB8.1.99 {ModbusAddress = 264; Command_write_byte = Force multiply coils (0x0f); Visibility = No}
  AT %QB8.1.99.0 [ByteOutput]
8 bit output module [ID2002] node 100, in %IB8.1.100 out %QB8.1.100 {ModbusAddress = 272; Command_write_byte = Force multiply coils (0x0f); Visibility = No}
  AT %QB8.1.100.0 [ByteOutput]
8 bit output module [ID2002] node 101, in %IB8.1.101 out %QB8.1.101 {ModbusAddress = 280; Command_write_byte = Force multiply coils (0x0f); Visibility = No}
  AT %QB8.1.101.0 [ByteOutput]
8 bit output module [ID2002] node 102, in %IB8.1.102 out %QB8.1.102 {ModbusAddress = 288; Command_write_byte = Force multiply coils (0x0f); Visibility = No}
  AT %QB8.1.102.0 [ByteOutput]
8 bit output module [ID2002] node 103, in %IB8.1.103 out %QB8.1.103 {ModbusAddress = 296; Command_write_byte = Force multiply coils (0x0f); Visibility = No}
  AT %QB8.1.103.0 [ByteOutput]
8 bit output module [ID2002] node 104, in %IB8.1.104 out %QB8.1.104 {ModbusAddress = 304; Command_write_byte = Force multiply coils (0x0f); Visibility = No}
  AT %QB8.1.104.0 [ByteOutput]
8 bit output module [ID2002] node 105, in %IB8.1.105 out %QB8.1.105 {ModbusAddress = 312; Command_write_byte = Force multiply coils (0x0f); Visibility = No}
  AT %QB8.1.105.0 [ByteOutput]
8 bit output module [ID2002] node 106, in %IB8.1.106 out %QB8.1.106 {ModbusAddress = 320; Command_write_byte = Force multiply coils (0x0f); Visibility = No}
  AT %QB8.1.106.0 [ByteOutput]
8 bit output module [ID2002] node 107, in %IB8.1.107 out %QB8.1.107 {ModbusAddress = 328; Command_write_byte = Force multiply coils (0x0f); Visibility = No}
  AT %QB8.1.107.0 [ByteOutput]
8 bit output module [ID2002] node 108, in %IB8.1.108 out %QB8.1.108 {ModbusAddress = 336; Command_write_byte = Force multiply coils (0x0f); Visibility = No}
  AT %QB8.1.108.0 [ByteOutput]
8 bit output module [ID2002] node 109, in %IB8.1.109 out %QB8.1.109 {ModbusAddress = 344; Command_write_byte = Force multiply coils (0x0f); Visibility = No}
  AT %QB8.1.109.0 [ByteOutput]
8 bit output module [ID2002] node 110, in %IB8.1.110 out %QB8.1.110 {ModbusAddress = 352; Command_write_byte = Force multiply coils (0x0f); Visibility = No}
  AT %QB8.1.110.0 [ByteOutput]
8 bit output module [ID2002] node 111, in %IB8.1.111 out %QB8.1.111 {ModbusAddress = 360; Command_write_byte = Force multiply coils (0x0f); Visibility = No}
  AT %QB8.1.111.0 [ByteOutput]
8 bit output module [ID2002] node 112, in %IB8.1.112 out %QB8.1.112 {ModbusAddress = 368; Command_write_byte = Force multiply coils (0x0f); Visibility = No}
  AT %QB8.1.112.0 [ByteOutput]
8 bit output module [ID2002] node 113, in %IB8.1.113 out %QB8.1.113 {ModbusAddress = 376; Command_write_byte = Force multiply coils (0x0f); Visibility = No}
  AT %QB8.1.113.0 [ByteOutput]
8 bit output module [ID2002] node 114, in %IB8.1.114 out %QB8.1.114 {ModbusAddress = 384; Command_write_byte = Force multiply coils (0x0f); Visibility = No}
  AT %QB8.1.114.0 [ByteOutput]
8 bit output module [ID2002] node 115, in %IB8.1.115 out %QB8.1.115 {ModbusAddress = 392; Command_write_byte = Force multiply coils (0x0f); Visibility = No}
  AT %QB8.1.115.0 [ByteOutput]
8 bit output module [ID2002] node 116, in %IB8.1.116 out %QB8.1.116 {ModbusAddress = 400; Command_write_byte = Force multiply coils (0x0f); Visibility = No}
  AT %QB8.1.116.0 [ByteOutput]
8 bit output module [ID2002] node 117, in %IB8.1.117 out %QB8.1.117 {ModbusAddress = 408; Command_write_byte = Force multiply coils (0x0f); Visibility = No}
  AT %QB8.1.117.0 [ByteOutput]
8 bit output module [ID2002] node 118, in %IB8.1.118 out %QB8.1.118 {ModbusAddress = 416; Command_write_byte = Force multiply coils (0x0f); Visibility = No}
  AT %QB8.1.118.0 [ByteOutput]
8 bit output module [ID2002] node 119, in %IB8.1.119 out %QB8.1.119 {ModbusAddress = 424; Command_write_byte = Force multiply coils (0x0f); Visibility = No}
  AT %QB8.1.119.0 [ByteOutput]
8 bit output module [ID2002] node 120, in %IB8.1.120 out %QB8.1.120 {ModbusAddress = 432; Command_write_byte = Force multiply coils (0x0f); Visibility = No}
  AT %QB8.1.120.0 [ByteOutput]
8 bit output module [ID2002] node 121, in %IB8.1.121 out %QB8.1.121 {ModbusAddress = 440; Command_write_byte = Force multiply coils (0x0f); Visibility = No}
  AT %QB8.1.121.0 [ByteOutput]
8 bit output module [ID2002] node 122, in %IB8.1.122 out %QB8.1.122 {ModbusAddress = 448; Command_write_byte = Force multiply coils (0x0f); Visibility = No}
  AT %QB8.1.122.0 [ByteOutput]
8 bit output module [ID2002] node 123, in %IB8.1.123 out %QB8.1.123 {ModbusAddress = 456; Command_write_byte = Force multiply coils (0x0f); Visibility = No}
  AT %QB8.1.123.0 [ByteOutput]
8 bit output module [ID2002] node 124, in %IB8.1.124 out %QB8.1.124 {ModbusAddress = 464; Command_write_byte = Force multiply coils (0x0f); Visibility = No}
  AT %QB8.1.124.0 [ByteOutput]
8 bit output module [ID2002] node 125, in %IB8.1.125 out %QB8.1.125 {ModbusAddress = 472; Command_write_byte = Force multiply coils (0x0f); Visibility = No}
  AT %QB8.1.125.0 [ByteOutput]
8 bit output module [ID2002] node 126, in %IB8.1.126 out %QB8.1.126 {ModbusAddress = 480; Command_write_byte = Force multiply coils (0x0f); Visibility = No}
  AT %QB8.1.126.0 [ByteOutput]
8 bit output module [ID2002] node 127, in %IB8.1.127 out %QB8.1.127 {ModbusAddress = 488; Command_write_byte = Force multiply coils (0x0f); Visibility = No}
  AT %QB8.1.127.0 [ByteOutput]
8 bit output module [ID2002] node 128, in %IB8.1.128 out %QB8.1.128 {ModbusAddress = 496; Command_write_byte = Force multiply coils (0x0f); Visibility = No}
  AT %QB8.1.128.0 [ByteOutput]
8 bit output module [ID2002] node 129, in %IB8.1.129 out %QB8.1.129 {ModbusAddress = 504; Command_write_byte = Force multiply coils (0x0f); Visibility = No}
  AT %QB8.1.129.0 [ByteOutput]
8 bit output module [ID2002] node 130, in %IB8.1.130 out %QB8.1.130 {ModbusAddress = 512; Command_write_byte = Force multiply coils (0x0f); Visibility = No}
  AT %QB8.1.130.0 [ByteOutput]
8 bit output module [ID2002] node 131, in %IB8.1.131 out %QB8.1.131 {ModbusAddress = 520; Command_write_byte = Force multiply coils (0x0f); Visibility = No}
  AT %QB8.1.131.0 [ByteOutput]
8 bit output module [ID2002] node 132, in %IB8.1.132 out %QB8.1.132 {ModbusAddress = 528; Command_write_byte = Force multiply coils (0x0f); Visibility = No}
  AT %QB8.1.132.0 [ByteOutput]
8 bit output module [ID2002] node 133, in %IB8.1.133 out %QB8.1.133 {ModbusAddress = 632; Command_write_byte = Force multiply coils (0x0f); Visibility = No}
  AT %QB8.1.133.0 [ByteOutput]
  AT %QB8.1.134.0 [ByteOutput]
AT %QB8.2.0 [ComChannel] Command (0xff - Start)
8 bit input module [ID2001] node 0, in %IB8.2.0 out %QB8.2.0 {ModbusAddress = 536; Command_read_byte = Read coils status (0x01); Visibility = No}
  AT %IB8.2.0.0 [ByteInput]
8 bit input module [ID2001] node 1, in %IB8.2.1 out %QB8.2.1 {ModbusAddress = 544; Command_read_byte = Read coils status (0x01); Visibility = No}
  AT %IB8.2.1.0 [ByteInput]
8 bit input module [ID2001] node 2, in %IB8.2.2 out %QB8.2.2 {ModbusAddress = 552; Command_read_byte = Read coils status (0x01); Visibility = No}
  AT %IB8.2.2.0 [ByteInput]
8 bit input module [ID2001] node 3, in %IB8.2.3 out %QB8.2.3 {ModbusAddress = 560; Command_read_byte = Read coils status (0x01); Visibility = No}
  AT %IB8.2.3.0 [ByteInput]
8 bit input module [ID2001] node 4, in %IB8.2.4 out %QB8.2.4 {ModbusAddress = 568; Command_read_byte = Read coils status (0x01); Visibility = No}
  AT %IB8.2.4.0 [ByteInput]
8 bit input module [ID2001] node 5, in %IB8.2.5 out %QB8.2.5 {ModbusAddress = 576; Command_read_byte = Read coils status (0x01); Visibility = No}
  AT %IB8.2.5.0 [ByteInput]
8 bit input module [ID2001] node 6, in %IB8.2.6 out %QB8.2.6 {ModbusAddress = 584; Command_read_byte = Read coils status (0x01); Visibility = No}
  AT %IB8.2.6.0 [ByteInput]
8 bit input module [ID2001] node 7, in %IB8.2.7 out %QB8.2.7 {ModbusAddress = 592; Command_read_byte = Read coils status (0x01); Visibility = No}
  AT %IB8.2.7.0 [ByteInput]
8 bit input module [ID2001] node 8, in %IB8.2.8 out %QB8.2.8 {ModbusAddress = 600; Command_read_byte = Read coils status (0x01); Visibility = No}
  AT %IB8.2.8.0 [ByteInput]
8 bit input module [ID2001] node 9, in %IB8.2.9 out %QB8.2.9 {ModbusAddress = 608; Command_read_byte = Read coils status (0x01); Visibility = No}
  AT %IB8.2.9.0 [ByteInput]
8 bit input module [ID2001] node 10, in %IB8.2.10 out %QB8.2.10 {ModbusAddress = 616; Command_read_byte = Read coils status (0x01); Visibility = No}
  AT %IB8.2.10.0 [ByteInput]
  AT %IB8.2.11.0 [ByteInput]
Real input module [ID2007] node 12, in %IB8.2.12 out %QB8.2.12 {ModbusAddress = 10256; Command_read_regs = Read holding Registers  (0x03); Visibility = No}
  panTimeToOpenCloseValve AT %ID8.2.12.0 [FloatInput]
Register input module [ID2003] node 13, in %IB8.2.13 out %QB8.2.13 {ModbusAddress = 10258; Command_read_regs = Read holding Registers  (0x03); Visibility = No}
  panMaxTemperature AT %IW8.2.13.0 [WordInput]
Register input module [ID2003] node 14, in %IB8.2.14 out %QB8.2.14 {ModbusAddress = 10259; Command_read_regs = Read holding Registers  (0x03); Visibility = No}
  panMinTemperature AT %IW8.2.14.0 [WordInput]
Real input module [ID2007] node 15, in %IB8.2.15 out %QB8.2.15 {ModbusAddress = 10260; Command_read_regs = Read holding Registers  (0x03); Visibility = No}
  panND0502setMaxDosVal AT %ID8.2.15.0 [FloatInput]
Real input module [ID2007] node 16, in %IB8.2.16 out %QB8.2.16 {ModbusAddress = 10262; Command_read_regs = Read holding Registers  (0x03); Visibility = No}
  panND0502setKoefProp AT %ID8.2.16.0 [FloatInput]
Real input module [ID2007] node 17, in %IB8.2.17 out %QB8.2.17 {ModbusAddress = 10264; Command_read_regs = Read holding Registers  (0x03); Visibility = No}
  panND0602setMaxDosVal AT %ID8.2.17.0 [FloatInput]
Real input module [ID2007] node 18, in %IB8.2.18 out %QB8.2.18 {ModbusAddress = 10266; Command_read_regs = Read holding Registers  (0x03); Visibility = No}
  panND0602setKoefProp AT %ID8.2.18.0 [FloatInput]
Real input module [ID2007] node 19, in %IB8.2.19 out %QB8.2.19 {ModbusAddress = 10268; Command_read_regs = Read holding Registers  (0x03); Visibility = No}
  panND0603setMaxDosVal AT %ID8.2.19.0 [FloatInput]
Real input module [ID2007] node 20, in %IB8.2.20 out %QB8.2.20 {ModbusAddress = 10270; Command_read_regs = Read holding Registers  (0x03); Visibility = No}
  panND0603setKoefProp AT %ID8.2.20.0 [FloatInput]
Real input module [ID2007] node 21, in %IB8.2.21 out %QB8.2.21 {ModbusAddress = 10272; Command_read_regs = Read holding Registers  (0x03); Visibility = No}
  panND0703pHsetValue AT %ID8.2.21.0 [FloatInput]
Real input module [ID2007] node 22, in %IB8.2.22 out %QB8.2.22 {ModbusAddress = 10274; Command_read_regs = Read holding Registers  (0x03); Visibility = No}
  panND0703YoutManual AT %ID8.2.22.0 [FloatInput]
Real input module [ID2007] node 23, in %IB8.2.23 out %QB8.2.23 {ModbusAddress = 10276; Command_read_regs = Read holding Registers  (0x03); Visibility = No}
  panND0703koeffI AT %ID8.2.23.0 [FloatInput]
Real input module [ID2007] node 24, in %IB8.2.24 out %QB8.2.24 {ModbusAddress = 10278; Command_read_regs = Read holding Registers  (0x03); Visibility = No}
  panND0703koeffD AT %ID8.2.24.0 [FloatInput]
Real input module [ID2007] node 25, in %IB8.2.25 out %QB8.2.25 {ModbusAddress = 10280; Command_read_regs = Read holding Registers  (0x03); Visibility = No}
  panND0703koeffP AT %ID8.2.25.0 [FloatInput]
Real input module [ID2007] node 26, in %IB8.2.26 out %QB8.2.26 {ModbusAddress = 10282; Command_read_regs = Read holding Registers  (0x03); Visibility = No}
  panND0803setMaxDosVal AT %ID8.2.26.0 [FloatInput]
Real input module [ID2007] node 27, in %IB8.2.27 out %QB8.2.27 {ModbusAddress = 10284; Command_read_regs = Read holding Registers  (0x03); Visibility = No}
  panND0803setKoefProp AT %ID8.2.27.0 [FloatInput]
Register input module [ID2003] node 28, in %IB8.2.28 out %QB8.2.28 {ModbusAddress = 10286; Command_read_regs = Read holding Registers  (0x03); Visibility = No}
  panND0804doseValue AT %IW8.2.28.0 [WordInput]
Real input module [ID2007] node 29, in %IB8.2.29 out %QB8.2.29 {ModbusAddress = 10287; Command_read_regs = Read holding Registers  (0x03); Visibility = No}
  panN0105flowSetValue AT %ID8.2.29.0 [FloatInput]
Real input module [ID2007] node 30, in %IB8.2.30 out %QB8.2.30 {ModbusAddress = 10289; Command_read_regs = Read holding Registers  (0x03); Visibility = No}
  panN0105YoutManual AT %ID8.2.30.0 [FloatInput]
Real input module [ID2007] node 31, in %IB8.2.31 out %QB8.2.31 {ModbusAddress = 10291; Command_read_regs = Read holding Registers  (0x03); Visibility = No}
  panN0105koeffI AT %ID8.2.31.0 [FloatInput]
Real input module [ID2007] node 32, in %IB8.2.32 out %QB8.2.32 {ModbusAddress = 10293; Command_read_regs = Read holding Registers  (0x03); Visibility = No}
  panN0105koeffD AT %ID8.2.32.0 [FloatInput]
Real input module [ID2007] node 33, in %IB8.2.33 out %QB8.2.33 {ModbusAddress = 10295; Command_read_regs = Read holding Registers  (0x03); Visibility = No}
  panN0105koeffP AT %ID8.2.33.0 [FloatInput]
Real input module [ID2007] node 34, in %IB8.2.34 out %QB8.2.34 {ModbusAddress = 10297; Command_read_regs = Read holding Registers  (0x03); Visibility = No}
  panFQS0301impulsValue AT %ID8.2.34.0 [FloatInput]
Real input module [ID2007] node 35, in %IB8.2.35 out %QB8.2.35 {ModbusAddress = 10299; Command_read_regs = Read holding Registers  (0x03); Visibility = No}
  panFQS0301correction AT %ID8.2.35.0 [FloatInput]
Real input module [ID2007] node 36, in %IB8.2.36 out %QB8.2.36 {ModbusAddress = 10301; Command_read_regs = Read holding Registers  (0x03); Visibility = No}
  panFPKtimeToWork AT %ID8.2.36.0 [FloatInput]
Real input module [ID2007] node 37, in %IB8.2.37 out %QB8.2.37 {ModbusAddress = 10303; Command_read_regs = Read holding Registers  (0x03); Visibility = No}
  panFPKnotStartedTime AT %ID8.2.37.0 [FloatInput]
Real input module [ID2007] node 38, in %IB8.2.38 out %QB8.2.38 {ModbusAddress = 10305; Command_read_regs = Read holding Registers  (0x03); Visibility = No}
  panFPKmaxPressureValue AT %ID8.2.38.0 [FloatInput]
Real input module [ID2007] node 39, in %IB8.2.39 out %QB8.2.39 {ModbusAddress = 10307; Command_read_regs = Read holding Registers  (0x03); Visibility = No}
  panFilterValueToRegen AT %ID8.2.39.0 [FloatInput]
ModBus (slave) [MODBUS_ID400] node 9, in %IB9 out %QB9 {SlaveIdentificator = 1; Visibility = No}
  Modbus [MODBUS_ID302] node 0, in %IB9.0 out %QB9.0
    TCP [TCP_ID221] node 0, in %IB9.0.0 out %QB9.0.0 {RemotePort = 502; Visibility = No}
  Float [Float] node 1, in %IB9.1 out %QB9.1
    remFT0101value AT %QD9.1.0 [FloatOutput] Расходомер на входе
  Float [Float] node 2, in %IB9.2 out %QB9.2
    remFQS0301totalAmount AT %QD9.2.0 [FloatOutput] Счетчик очищенных стоков
  Float [Float] node 3, in %IB9.3 out %QB9.3
    remTemperatureValue AT %QD9.3.0 [FloatOutput] Температура в помещении
  8 bits [8Bit] node 4, in %IB9.4 out %QB9.4
    AT %QB9.4.0 [ByteOutput]
  8 bits [8Bit] node 5, in %IB9.5 out %QB9.5
    AT %QB9.5.0 [ByteOutput]
*)

(* Global variable list: Global_Variables *)
VAR_GLOBAL
	wordMaxValue: WORD := 65535;		(*max value of WORD.*)
END_VAR

(* POU PLC_PRG, CFC *)
PROGRAM PLC_PRG
VAR
	rTrigStartInitializer: R_TRIG;		(*Детектор переднего фронта,
			инициализирует булевы переменные при старте программы.*)
	startInitializer: BOOL;		(*Инициализирует булевы переменные при старте программы.*)

	temperatureLimits: LIMITALARM;		(*блок контроля границ допустимой температуры в помещении*)
	alarmHighTemperature: BOOL;		(*температура выше заданного диапазона*)
	alarmLowTemperature: BOOL;		(*температура ниже заданного диапазона*)
	temperatureValue: REAL;		(*значение температуры в помещении*)
	DD1_AI0_temperature: DECODE_FLOAT;		(*блок контроля состояния аналогового входа ПЛК для датчика температуры в помещении*)
	DD1_AI1_flow: DECODE_FLOAT;		(*блок контроля состояния аналогового входа ПЛК для расходомера FT01.01*)

	ND0502dosing: DosingPumpProportional;		(*Блок управления дозированием насосов НД05.02/01 и НД05.02/02.
			Пропорционально расходу по FT01.01*)
	ND0502regime: choosePumpRegime;		(*Блок выбора режима включения НД05.02/01 и НД05.02/02.*)
	ND0502manager: TwoPumpManager;		(*Блок управления включением дозирующих насосов
			НД05.02/01 и НД05.02/02.*)

	ND0602dosing: DosingPumpProportional;		(*Блок управления дозированием насосов НД06.02/01 и НД06.02/02.
			Пропорционально расходу по FT01.02.*)
	ND0602regime: choosePumpRegime;		(*Блок выбора режима включения НД06.02/01 и НД06.02/02.*)
	ND0602manager: TwoPumpManager;		(*Блок управления включением дозирующих насосов
			НД06.02/01 и НД06.02/02.*)

	ND0603dosing: DosingPumpProportional;		(*Блок управления дозированием насосов НД06.03/01 и НД06.03/02.
						Пропорционально расходу по FT01.01*)
	ND0603regime: choosePumpRegime;		(*Блок выбора режима включения НД06.03/01 и НД06.03/02.*)
	ND0603manager: TwoPumpManager;		(*Блок управления включением дозирующих насосов
						НД06.03/01 и НД06.03/02.*)

	ND0703pidReg: PID;		(*Блок автоматического поддержания заданного значения рН стоков подачей щелочи через НД07.03
								по показаниям QE01.01.*)
	ND0703regime: choosePumpRegime;		(*Блок выбора режима включения НД07.03/01 и НД07.03/02.*)
	ND0703manager: TwoPumpManager;		(*Блок управления включением дозирующих насосов
									НД07.03/01 и НД07.03/02*)

	ND0803dosing: DosingPumpProportional;		(*Блок управления дозированием насосов НД08.03*)
	ND0803regime: choosePumpRegime;		(*Блок выбора режима включения насосов НД08.03.*)
	ND0803manager: TwoPumpManager;		(*Блок управления включением дозирующих насосов НД08.03.*)

	ND0804linearTransformator: LIN_TRAFO;		(*Блок преобразования сигнала на управление от 0 до 100% в 4...20мА*)

	DD1_AI1_FT0101: DECODE_FLOAT;		(*Блок контроля аналогового входа DD1_AI1 (расходомер FT01.01)*)
	DD1_AI2_FT0102: DECODE_FLOAT;		(*блок контроля состояния аналогового входа ПЛК для расходомера FT01.02*)
	DD1_AI3_QE0101: DECODE_FLOAT;		(*блок контроля состояния аналогового входа ПЛК для рН-метра QE01.01*)
	DD1_AI4_QE0102: DECODE_FLOAT;		(*блок контроля состояния аналогового входа ПЛК для рН-метра QE01.02*)

	DD1_AI1_FT0101value: REAL;		(*Показания расходомера FT01.01 после блока контроля аналогового входа ПЛК.*)
	DD1_AI2_FT0102value: REAL;		(*Показания расходомера FT01.02 после блока контроля аналогового входа ПЛК.*)
	DD1_AI3_QE0101value: REAL;		(*Показания рН-метра QE01.01 после блока контроля аналогового входа ПЛК.*)
	DD1_AI4_QE0102value: REAL;		(*Показания рН-метра QE01.02 после блока контроля аналогового входа ПЛК*)

	N0105regime: choosePumpRegime;		(*Блок выбора режима включения Н05.01*)
	N0105twoPumpOneDriveManager: TwoPumpOneDriveManager;		(*блок управления двумя насосами от одного частотника*)
	N0105pidReg: PID;		(*Блок автоматического поддержания заданного значения расхода по показаниям FT01.02*)

	N010501alarm: BOOL;		(*Авария насоса Н01.05/01*)
	N010502alarm: BOOL;		(*Авария насоса Н01.05/02*)
	N0105minFlow: REAL := 10;		(*Минимальное значение расхода. Если при включенном насосе расход меньше = авария.
			По умолчанию, если ничего не подключено ко входу, равно 10 кубометров в час.*)

	N010501alarmTrig: RS;		(*Триггер защелка аварии Н01.05/01.*)
	N010502alarmTrig: RS;		(*Триггер защелка аварии Н01.05/02.*)
	N0105timerminFlow: TON;		(*Таймер контроля времени на создание потока включенным насосом.*)
	N0105startTrigg: RS;		(*Триггер защелкивающий условие для старта насоса, и сбрасывающий старт при сухом ходе.*)

	N0105startTrig: R_TRIG;		(*Ловит передний фронт включения от кнопки для запуска насоса.*)
	N0105stopTrig: F_TRIG;		(*Ловит спад сигнала, значит нажата кнопка СТОП.*)
	N0105regByCinit: R_TRIG;		(*Детектор переднего фронта выбора режима по кол-ву вкл.*)
	N0105regWTinit: R_TRIG;		(*Детектор переднего фронта выбора режима по наработке.*)
	N0105regByCtrig: RS;		(*Защелка выбора режима по кол-ву включ.*)
	N0105regWTtrig: RS;		(*Защелка выбора режима по наработке.*)

	N0105statStartedP1: BOOL;	(*Статус - запуск первого насоса Н01.05/01*)
	N0105statStartedP2: BOOL;	(*Статус - запуск второго насоса Н01.05/02*)

	ZDE0225: SimpleValve;		(*Управление заслонкой ЗДЭ02.25 (наполнение РЧВ02.03)*)
	ZDE0225errorToOpen: BOOL;		(*Авария на открытие ЗДЭ02.25 (не открылась за заданное время).*)
	ZDE0225errorToClose: BOOL;		(*Авария на закрытие ЗДЭ02.25 (не закрылась за заданное время).*)

	FPKstartTrig: RS;		(*Триггер сигнала запуска фильтр-пресса.*)
	FPKstopTimer: TOF;		(*Таймер задержки сигнала на останов фильтр-пресса
			(после спада сигнала уровня осадка).*)
	FPKstopFtrig: F_TRIG;		(*Детектор спада сигнала от таймера останова ФПК
			для подачи сигнала на останов.*)
	DD1_AI5_FPK: DECODE_FLOAT;		(*контроль входа AI6 контроллера на обрыв (давление от фильтр-пресса).*)
	DD1_AI5_FPKpressureValue: REAL;		(*Давление на входе в ФПК,
			сигнал после блока контроля входа на обрыв.*)
	FPKnotStartedTimer: TON;		(*Таймер задержки после подачи сигнала на запуск ФПК
			о том, что он не запустился. *)
	FPKnotStarted: BOOL;		(*Сигнал, что ФПК не запустился спустя заданное время после подачи
			на него сигнала на старт.*)
	FPKneedToClean: BOOL;		(*Необходимо почистить ФПК!*)
	FPKneedToCleanTrig: RS;		(*Триггер сигнала о том, что нужно почистить ФПК.*)
	FPKneedToCleanReset: BOOL;		(*Сброс сигнала о необходимости очистки ФПК.*)
	FPKneedToCleanResetFtrig: F_TRIG;		(*Детектор спада сигнала на сброс сигнала о грязном фильтр-прессе.*)
	FPKneedToCleanResetRtrig: R_TRIG;		(*Детектор фронта сигнала на сброс необходимости чистить фильтр пресс.*)

	FPKkshe0401: SimpleValve;		(*Блок управления клапаном КШЭ04.01 перед ФПК.*)
	FPKkshe0401errorToOpen: BOOL;		(*Авария на открытие КШЭ04.01*)
	FPKkshe0401errorToClose: BOOL;		(*Авария на закрытие КШЭ04.01*)
	FPKkshe0401DelayToOpen: TON;		(*Задержка на открытие, чтобы не сработало одновременно с закрытием.*)
	FPKkshe0401DelayToClose: TON;		(*Задержка на закрытие, чтобы не сработало одновременно с открытием.*)

	N0404twoPumpManager: TwoPumpManager;		(*Блок управления дренажными насосами Н04.04*)
	N0401choosePumpRegime: choosePumpRegime;		(*Блок выбора режима работы дренажных насосов Н04.04.*)

	UFO0301manager: TwoPumpManager;		(*Блок управления включением УФО 03.01 в зависимости от выбранного режима.*)
	UFO0301regimeManager: choosePumpRegime;		(*Блок выбора режима работы УФО 03.01.*)
	UFO0301startDelay: TON;		(*Таймер задержки на включение после появления стоков в расходомере FT01.02*)

	FQS0301rTrig: R_TRIG;		(*Детектор переднего фронта импульсного счетчика расходомера.*)
	FQS0301resetRtrig: R_TRIG;		(*Детектор переднего фронта на сброс значений счетчика.*)
	FQS0301addCorrRtrig: R_TRIG;		(*Детектор переднего фронта сигнала на прибавку коррекции.*)
	FQS0301deleteCorrRtrig: R_TRIG;		(*Детектор переднего фронта сигнала на вычитание коррекции.*)

	N0204chooseRegime: choosePumpRegime;		(*Блок управления выбора режима работы насосов Н02.04*)
	N0204manager: TwoPumpManager;		(*Блок управления работой насосов Н02.04.*)
	N020401fTrigStop: F_TRIG;		(*Детектор спада сигнала на включение насоса Н02.04/01 для сброса самоподхвата реле.*)
	N020402fTrigStop: F_TRIG;		(*Детектор спада сигнала на включение насоса Н02.04/02 для сброса самоподхвата реле.*)
	N0204stop: TOF;		(*таймер удержания сигнала на выключение насосов Н02.04 для гарантированного отключения реле.*)

	filterPulserGen: PulsePerSec;		(*Генератор импульсов каждую секунду для подсчета суммарного
			объема стоков через FT01.02.*)
	filterTotalAmountReset: BOOL;		(*Сброс наработки счетчика FT01.02, начало нового отсчета до
			следующей регенерации.*)
	filterFailToRegen020101: BOOL;		(*Не удалось запустить регенерацию (промывку) ФС02.01/01.*)
	filterFailToRegen020102: BOOL;		(*Не удалось запустить регенерацию (промывку) ФС02.01/02.*)
	FS0201manager: FilterQueueManager;		(*блок управления промывкой ФС02.01*)
	ZD0201: SimpleValve;		(*Блок управления задвижкой 02.01*)
	ZD0207: SimpleValve;		(*блок управления задвижкой 02.07*)
	alarmZD020107: BOOL;		(*авария задвижки 02.01 или 02.07 на открытие или закрытие.*)
	filterStartNewQueue: BOOL;		(*Начать новую очередь промывки фильтров.*)
	regeneratedFS0201: BOOL;		(*Статус - фильтр ФС02.01 промыт*)
	FS020101manager: FilterQueueManager;		(*блок управления промывкой ФС02.01/01*)
	FS020102manager: FilterQueueManager;		(*Блок управления промывкой фильтра ФС02.01/02*)
	ZD0202: SimpleValve;		(*Блок управления задвижкой ЗДЭ02.02*)
	ZD0208: SimpleValve;		(*Блок управления задвижкой ЗДЭ02.08*)
	alarmZD020208: BOOL;		(*авария на открытие или закрытие ЗДЭ02.02 или ЗДЭ02.08.*)
	regeneratedFS020101: BOOL;		(*Статус - фильтр ФС02.01/01 промыт*)
	regeneratedFS020102: BOOL;		(*Статус - фильтр ФС02.01/02 промыт.*)
	FS020103manager: FilterQueueManager;		(*блок управления промывкой фильтра ФС02.01/03*)
	ZD0203: SimpleValve;		(*блок управления ЗДЭ02.03*)
	ZD0209: SimpleValve;		(*блок управления ЗДЭ02.09*)
	alarmZD020309: BOOL;		(*авария на открытие или закрытие ЗДЭ02.03 или ЗДЭ02.09.*)
	regeneratedFS020103: BOOL;		(*Фильтр ФС02.01/03 промыт в этой сессии очереди.*)
	filterFailToRegen020103: BOOL;		(*Не удалось запустить регенерацию ФС02.01/03*)
	FS020104manager: FilterQueueManager;		(*блок управления промывкой фильтра ФС02.01/04.*)
	ZD0204: SimpleValve;		(*блок управления ЗДЭ02.04*)
	ZD0210: SimpleValve;		(*блок управления ЗДЭ02.10*)
	alarmZD020410: BOOL;		(*авария на открытие или закрытие ЗДЭ02.04 или ЗДЭ02.10*)
	regeneratedFS020104: BOOL;		(*Фильтр ФС02.01/04 промыт*)
	filterFailToRegen020104: BOOL;		(*Не удалось запустить регенерацию ФС02.01/04*)
	errorToOpenZD0210: BOOL;		(*Не удалось открыть ЗДЭ02.10*)
	FS020105manager: FilterQueueManager;		(*блок управления промывкой фильтра ФС02.01/04*)
	ZD0205: SimpleValve;		(*блок управления ЗДЭ02.05*)
	ZD0211: SimpleValve;		(*блок управления ЗДЭ02.11*)
	alarmZD020511: BOOL;		(*авария на открытие или закрытие ЗДЭ02.05 или ЗДЭ02.11*)
	regeneratedFS020105: BOOL;		(*Фильтр ФС02.01/05 промыт*)
	filterFailToRegen020105: BOOL;		(*Не удалось запустить регенерацию ФС02.01/05*)
	FS020106manager: FilterQueueManager;		(*блок управления промывкой ФС02.01/06*)
	ZD0206: SimpleValve;		(*блок управления ЗДЭ02.06*)
	ZD0212: SimpleValve;		(*блок управления ЗДЭ02.12*)
	alarmZD020612: BOOL;		(*авария на открытие или закрытие ЗДЭ02.06 или 02.12*)
	FS020201manager: FilterQueueManager;		(*блок управления промывкой ФС02.02/01*)
	ZD0213: SimpleValve;		(*блок управления ЗДЭ02.13*)
	ZD0219: SimpleValve;		(*блок управления ЗДЭ02.19*)
	alarmZD021319: BOOL;		(*авария на открытие или закрытие ЗДЭ02.13 или ЗДЭ02.19*)
	regeneratedFS020201: BOOL;		(*Фильтр ФС02.02/01 промыт*)
	filterFailToRegen020201: BOOL;		(*Не удалось запустить регенерацию ФС02.02/01*)
	FS020202manager: FilterQueueManager;		(*блок управления промывкой ФС02.02/02*)
	ZD0214: SimpleValve;		(*блок управления ЗДЭ02.14*)
	ZD0220: SimpleValve;		(*блок управления ЗДЭ02.20*)
	alarmZD021420: BOOL;		(*авария на открытие или на закрытие ЗДЭ02.14 или ЗДЭ02.20*)
	regeneratedFS020202: BOOL;		(*Фильтр ФС02.02/02 промыт *)
	filterFailToRegen020202: BOOL;		(*Не удалось запустить регенерацию ФС02.02/02*)
	FS020203manager: FilterQueueManager;		(*блок управления ФС02.02/03*)
	ZD0215: SimpleValve;		(*блок управления ЗДЭ02.15*)
	ZD0221: SimpleValve;		(*блок управления ЗДЭ02.21*)
	regeneratedFS020203: BOOL;		(*Фильтр ФС02.02/03 промыт в этой сессии очереди.*)
	filterFailToRegen020203: BOOL;		(*Не удалось запустить регенерацию ФС02.02/03*)
	alarmZD021521: BOOL;		(*авария на открытие или на закрытие ЗДЭ02.15 или ЗДЭ02.21*)
	alarmZD021622: BOOL;		(*авария на открытие или на закрытие ЗДЭ02.16 или ЗДЭ 02.22*)
	FS020204manager: FilterQueueManager;		(*блок управления промывкой ФС02.02/04*)
	ZD0216: SimpleValve;		(*блок управления ЗДЭ02.16*)
	ZD0222: SimpleValve;		(*блок управления ЗДЭ02.22*)
	regeneratedFS020204: BOOL;		(*Фильтр ФС02.02/04 промыт*)
	filterFailToRegen020204: BOOL;		(*Не удалось запустить регенерацию ФС02.02/04*)
	FS020205manager: FilterQueueManager;		(*блок управления ФС02.02/05*)
	ZD0217: SimpleValve;		(*блок управления ЗДЭ02.17*)
	ZD0223: SimpleValve;		(*блок управления ЗДЭ02.23*)
	regeneratedFS020205: BOOL;		(*Фильтр ФС02.02/05 промыт*)
	filterFailToRegen020205: BOOL;		(*Не удалось запустить регенерацию ФС02.02/05*)
	alarmZD021723: BOOL;		(*авария на открытие или на закрытие ЗДЭ02.17 или ЗДЭ02.24*)
	FS020206manager: FilterQueueManager;		(*блок управления промывкой ФС02.02/06*)
	ZD0218: SimpleValve;		(*блок управления ЗДЭ02.18*)
	ZD0224: SimpleValve;		(*блок управления ЗДЭ02.24*)
	alarmZD021824: BOOL;		(*авария на открытие или на закрытие ЗДЭ02.18 или ЗДЭ02.24*)
	regeneratedFS020206: BOOL;		(*Фильтр ФС02.02/06 промыт *)
	filterFailToRegen020206: BOOL;		(*Не удалось запустить регенерацию ФС02.02/06*)
	filterFailToRegen020106: BOOL;		(*Не удалось запустить регенерацию ФС02.01/06*)

	alarmPLKnetwork: BOOL;		(*Авария сети ПЛК.
			Скорее всего - обрыв или ошибка в каком-то из модулей.*)
	alarmPLKnetworkDelay: TOF;		(*Задержка формирования аварии сети ПЛК.
			По умолчанию = 20 секунд.*)

	alarmND050201: BOOL;
	alarmND050202: BOOL;
	alarmND060201: BOOL;
	alarmND060202: BOOL;
	alarmND060301: BOOL;
	alarmND060302: BOOL;
	alarmND070301: BOOL;
	alarmND070302: BOOL;
	alarmND080301: BOOL;
	alarmND080302: BOOL;
	alarmND0804: BOOL;
	alarmOGM0104overload: BOOL;
	alarmZDE0225power: BOOL;
	alarmRCHV0203overload: BOOL;
	alarmN040402: BOOL;
	alarmN040401: BOOL;
	alarmM0604: BOOL;
	alarmM0702: BOOL;
	alarmM0802: BOOL;
	alarmN020401: BOOL;
	alarmN020402: BOOL;
	alarmFS020101: BOOL;
	alarmFS020102: BOOL;
	alarmFS020103: BOOL;
	alarmFS020104: BOOL;
	alarmFS020105: BOOL;
	alarmFS020106: BOOL;
	alarmFS020201: BOOL;
	alarmFS020202: BOOL;
	alarmFS020203: BOOL;
	alarmFS020204: BOOL;
	alarmFS020205: BOOL;
	alarmFS020206: BOOL;
	alarmZDE0201power: BOOL;
	alarmZDE0202power: BOOL;
	alarmZDE0203power: BOOL;
	alarmZDE0204power: BOOL;
	alarmZDE0205power: BOOL;
	alarmZDE0206power: BOOL;
	alarmZDE0207power: BOOL;
	alarmZDE0208power: BOOL;
	alarmZDE0209power: BOOL;
	alarmZDE0210power: BOOL;
	alarmZDE0211power: BOOL;
	alarmZDE0212power: BOOL;
	alarmZDE0213power: BOOL;
	alarmZDE0214power: BOOL;
	alarmZDE0215power: BOOL;
	alarmZDE0216power: BOOL;
	alarmZDE0217power: BOOL;
	alarmZDE0218power: BOOL;
	alarmZDE0219power: BOOL;
	alarmZDE0220power: BOOL;
	alarmZDE0221power: BOOL;
	alarmZDE0222power: BOOL;
	alarmZDE0223power: BOOL;
	alarmZDE0224power: BOOL;
	alarmKNS: BOOL;
	alarmPowerSocketFS: BOOL;
	alarmKEMvalvesPower: BOOL;
	alarmEmergencyPressed: BOOL;
	alarmRKF: BOOL;
	alarm: BOOL;		(*Общая авария*)
	alarmKSHE0401power: BOOL;
	workTimeND050201: TimeFromWorkTime;		(*Наработка НД05.02/01*)
	workTimeND050202: TimeFromWorkTime;		(*Наработка НД05.02/02*)
	workTimeND060201: TimeFromWorkTime;		(*Наработка НД06.02/01*)
	workTimeND060202: TimeFromWorkTime;		(*Наработка НД06.02/02*)
	workTimeND060301: TimeFromWorkTime;		(*Наработка НД06.03/01*)
	workTimeND060302: TimeFromWorkTime;		(*Наработка НД06.03/02*)
	workTimeND070301: TimeFromWorkTime;		(*Наработка НД07.03/01*)
	workTimeND070302: TimeFromWorkTime;		(*Наработка НД07.03/02*)
	workTimeND080301: TimeFromWorkTime;		(*Наработка НД08.03/01*)
	workTimeND080302: TimeFromWorkTime;		(*Наработка НД08.03/02*)
	workTimeN010501: TimeFromWorkTime;		(*Наработка Н01.05/01*)
	workTimeN010502: TimeFromWorkTime;		(*Наработка Н01.05/02*)
	workTimeN020401: TimeFromWorkTime;		(*Наработка Н02.04/01*)
	workTimeN020402: TimeFromWorkTime;		(*Наработка Н02.04/02*)
	workTimeN040401: TimeFromWorkTime;		(*Наработка Н04.04/01*)
	workTimeN040402: TimeFromWorkTime;		(*Наработка Н04.04/02*)
	workTimeUFO030101: TimeFromWorkTime;		(*Наработка УФО03.01/01*)
	workTimeUFO030102: TimeFromWorkTime;		(*Наработка УФО03.01/02*)
	testKSHE0401: BOOL;		(*Тест задвижки КШЭ04.01.
			имитация сигнала работы ФПК.*)
	testZDE0225: BOOL;		(*Тест ЗДЭ02.25
			имитация сигнала раб.уровня (1 = норма, ЗДЭ закрыт).*)
	ZDE0301: SimpleValve;
	ZDE0302: SimpleValve;
	errorToOpenZDE0301: BOOL;		(*ЗДЭ03.01 не открылась за заданное время.*)
	errorToCloseZDE0301: BOOL;		(*ЗДЭ03.01 не закрылась за заданное время.*)
	errorToOpenZDE0302: BOOL;		(*ЗДЭ03.02 не открылась за заданное время.*)
	errorToCloseZDE0302: BOOL;		(*ЗДЭ03.02 не закрылась за заданное время.*)
	alarmZDE0301power: BOOL;		(*сработал автомат ЗДЭ03.01*)
	alarmZDE0302power: BOOL;		(*сработал автомат ЗДЭ03.02*)
	manualZDE0301: BOOL;		(*Ручное открытие/закрытие ЗДЭ03.01*)
	manualZDE0302: BOOL;		(*Ручное открытие/закрытие ЗДЭ03.02*)
	testZDE03: BOOL;		(*Режим тестирования ЗДЭ03.01 и ЗДЭ03.02.
			В этом режиме автоматический пуск УФО от ПЛК невозможен!*)
	UFO030101startTrig: R_TRIG;		(*Триггер переднего фронта на старт УФО03.01/01*)
	UFO030102startTrig: R_TRIG;		(*Триггер переднего фронта на старт УФО03.01/02.*)
	UFO030101stopTrig: F_TRIG;		(*Триггер заднего фронта (спад сигнала) на останов УФО03.01/01.*)
	UFO030102stopTrig: F_TRIG;		(*Триггер заднего фронта (спад сигнала) на останов УФО03.01/02.*)

	volumeToRegen: REAL;		(*Объем стоков до следующей регенерации (заданный минус текущий накопленный
			через ЭМР FT01.02)*)
	linTrafND050201: LIN_TRAFO;
	linTraf060201: LIN_TRAFO;
	linTraf060202: LIN_TRAFO;
	linTraf060301: LIN_TRAFO;
	linTraf060302: LIN_TRAFO;
END_VAR
VAR_INPUT
	alarmReset: BOOL;		(*Сброс аварий.*)

	ND0502resetCountP1: BOOL;		(*Сбросить счетчик количества включений НД05.02/01.*)
	ND0502resetCountP2: BOOL;		(*Сбросить счетчик количества включений НД05.02/02.*)
	ND0502resetWorkTimeP1: BOOL;		(*Сбросить счетчик наработки НД05.02/01.*)
	ND0502resetWorkTimeP2: BOOL;		(*Сбросить счетчик наработки НД05.02/02.*)

	ND0602resetCountP1: BOOL;		(*Сбросить счетчик количества включений НД06.02/01.*)
	ND0602resetCountP2: BOOL;		(*Сбросить счетчик количества включений НД06.02/02.*)
	ND0602resetWorkTimeP1: BOOL;		(*Сбросить счетчик количества наработки НД06.02/01.*)
	ND0602resetWorkTimeP2: BOOL;		(*Сбросить счетчик количества наработки НД06.02/02.*)

	ND0603resetCountP1: BOOL;		(*Сбросить счетчик количества включений НД06.03/01.*)
	ND0603resetCountP2: BOOL;		(*Сбросить счетчик количества включений НД06.03/02.*)
	ND0603resetWorkTimeP1: BOOL;		(*Сбросить счетчик времени наработки НД06.03/01.*)
	ND0603resetWorkTimeP2: BOOL;		(*Сбросить счетчик времени наработки НД06.03/02.*)

	ND0703resetCountP1: BOOL;		(*Сбросить счетчик количества включений НД07.03/01.*)
	ND0703resetCountP2: BOOL;		(*Сбросить счетчик количества включений НД07.03/02.*)
	ND0703resetWorkTimeP1: BOOL;		(*Сбросить счетчик наработки НД07.03/01.*)
	ND0703resetWorkTimeP2: BOOL;		(*Сбросить счетчик наработки НД07.03/02.*)
	ND0703YoutManual: REAL;		(*Задание значения выходу Y в ручном режиме (4...20мА).*)
	ND0703YmanAuto: BOOL;		(*Выбор управления выходом Y в ручном или автоматическом режиме.*)

	ND0803resetCountP1: BOOL;		(*Сброс счетчика количества включений НД08.03/01.*)
	ND0803resetCountP2: BOOL;		(*Сброс счетчика количества включений НД08.03/02.*)
	ND0803resetWorkTimeP1: BOOL;		(*Сброс счетчика наработки НД08.03/01.*)
	ND0803resetWorkTimeP2: BOOL;		(*Сброс счетчика наработки НД08.03/02.*)

	N0105YoutManual: REAL;		(*Задание значения выходу Y в ручном режиме (4...20мА).*)
	N0105YmanAuto: BOOL;		(*Выбор управления выходом Y в ручном или автоматическом режиме.*)
	N0105resetCountP1: BOOL;		(*Сброс счетчика количества включений Н01.05/01.*)
	N0105resetCountP2: BOOL;		(*Сброс счетчика количества включений Н01.05/02.*)
	N0105resetWorkTimeP1: BOOL;		(*Сброс счетчика наработки Н01.05/01.*)
	N0105resetWorkTimeP2: BOOL;		(*Сброс счетчика наработки Н01.05/02.*)

	N0404resetCountP1: BOOL;		(*Сброс счетчика количества включений Н04.04/01.*)
	N0404resetCountP2: BOOL;		(*Сброс счетчика количества включений Н04.04/02.*)
	N0404resetWorkTimeP1: BOOL;		(*Сброс счетчика времени наработки Н04.04/01.*)
	N0404resetWorkTimeP2: BOOL;		(*Сброс счетчика времени наработки Н04.04/02.*)

	UFO0301resetCountP1: BOOL;		(*Сброс счетчика количества включений УФО: 03.01/01.*)
	UFO0301resetCountP2: BOOL;		(*Сброс счетчика количества включений УФО: 03.01/02.*)
	UFO0301resetWorkTimeP1: BOOL;		(*Сброс счетчика наработки УФО: 03.01/01.*)
	UFO0301resetWorkTimeP2: BOOL;		(*Сброс счетчика наработки УФО: 03.01/02.*)

	FQS0301reset: BOOL;		(*Сброс накопленного счетчиком значения.*)
	FQS0301correction: REAL;		(*Коррекция показаний счетчика.*)
	FQS0301addCorrection: BOOL;		(*Прибавить введенную коррекцию к накопленной сумме стоков.*)
	FQS0301deleteCorrection: BOOL;		(*Вычесть введенную коррекцию из накопленной суммы стоков.*)

	N0204resetCountP1: BOOL;		(*Сброс счетчика количества включений Н02.04/01.*)
	N0204resetCountP2: BOOL;		(*Сброс счетчика количества включений Н02.04/02.*)
	N0204resetWorkTimeP1: BOOL;		(*Сброс счетчика наработки Н02.04/01.*)
	N0204resetWorkTimeP2: BOOL;		(*Сброс счетчика наработки Н02.04/02.*)

END_VAR
VAR_OUTPUT
	ND0502dosingError: BOOL;		(*Ошибка дозирования НД05.02.
			Проверить заданные уставки.*)
	ND0502statRegimeP1M: BOOL;		(*статус: режим НД05.02 - насос 1 = главный.*)
	ND0502statRegimeP2M: BOOL;		(*статус: режим НД05.02 - насос 2 = главный*)
	ND0502statRegimeByC: BOOL;		(*статус: режим НД05.02 - по количеству включений*)
	ND0502statRegimeByWT: BOOL;		(*статус: режим НД05.02 - по наработке*)

	ND0602dosingError: BOOL;		(*Ошибка дозирования НД06.02/01-02.
						Проверить заданные уставки.*)
	ND0602statRegimeP1M: BOOL;		(*статус: режим НД0602 - насос 1 = главный.*)
	ND0602statRegimeP2M: BOOL;		(*статус: режим НД06.02 - насос 2 = главный.*)
	ND0602statRegimeByC: BOOL;		(*статус: режим НД06.02 - по количеству включений.*)
	ND0602statRegimeByWT: BOOL;		(*статус: режим НД06.02 - по наработке.*)

	ND0603dosingError: BOOL;		(*Ошибка дозирования НД06.03.
						Проверить заданные уставки.*)
	ND0603statRegimeP1M: BOOL;		(*статус: режим НД0603 - насос 1 = главный.*)
	ND0603statRegimeP2M: BOOL;		(*статус: режим НД0603 - насос 2 = главный.*)
	ND0603statRegimeByC: BOOL;		(*статус: режим НД06.03 - по количеству включений.*)
	ND0603statRegimeByWT: BOOL;		(*статус: режим НД06.03 - по наработке.*)

	ND0703statRegimeP1M: BOOL;		(*статус: режим НД0703 - насос 1 = главный.*)
	ND0703statRegimeP2M: BOOL;		(*статус: режим НД0703 - насос 2 = главный.*)
	ND0703statRegimeByC: BOOL;		(*статус: режим НД07.03 - по количеству включений.*)
	ND0703statRegimeByWT: BOOL;		(*статус: режим НД07.03 - по наработке.*)

	ND0803dosingError: BOOL;		(*Ошибка блока дозирования НД08.03.*)
	ND0803statRegimeP1M: BOOL;		(*статус: режим НД08.03 - насос 1 = главный*)
	ND0803statRegimeP2M: BOOL;		(*статус: режим НД08.03 - насос 2 = главный*)
	ND0803statRegimeByC: BOOL;		(*статус: режим НД08.03 - по количеству включений*)
	ND0803statRegimeByWT: BOOL;		(*статус: режим НД08.03 - по наработке.*)

	ND0804dosingError: BOOL;		(*Ошибка дозирования НД08.04. Проверь уставки.*)

	DD1_AI0_error: BOOL;		(*авария входа AI1 (возможно, обрыв)*)
	DD1_AI1_error: BOOL;		(*авария входа AI2 (возможно, обрыв)*)
	DD1_AI2_error: BOOL;		(*авария входа AI3 (возможно, обрыв)*)
	DD1_AI3_error: BOOL;		(*авария входа AI4 (возможно, обрыв)*)
	DD1_AI4_error: BOOL;		(*авария входа AI5 (возможно, обрыв)*)

	N0105statRegimeP1M: BOOL;		(*статус: режим Н01.05/01 = главный.*)
	N0105statRegimeP2M: BOOL;		(*статус: режим Н01.05/02 = главный.*)
	N0105statRegimeByC: BOOL;		(*статус: режим Н01.05 = по количеству включений.*)
	N0105statRegimeByWT: BOOL;		(*статус: режим Н01.05 = по наработке.*)

	DD1_AI5_error: BOOL;		(*Авария входа AI6 ПЛК.
			ВОзможно - обрыв.*)

	N0404statRegimeP1M: BOOL;		(*Статус: активен режим - главный насос Н04.04/01.*)
	N0404statRegimeP2M: BOOL;		(*Статус: активен режим - главный насос Н04.04/02.*)
	N0404statRegimeByC: BOOL;		(*Статус: активен режим - по количеству включений.*)
	N0404statRegimeWT: BOOL;		(*Статус: активен режим - по наработке.*)

	UFO0301statRegimeP1M: BOOL;		(*Статус: режим главный насос УФО: 03.01/01*)
	UFO0301statRegimeP2M: BOOL;		(*Статус: режим главный насос УФО: 03.01/02*)
	UFO0301statRegimeByC: BOOL;		(*Статус: режим УФО по количеству включений*)
	UFO0301statRegimeWT: BOOL;		(*Статус: режим УФО по наработке*)
	UFO0301noFlowAttention: BOOL;		(*Переменная появления предостережения, что УФО включена в ручном режиме,
			когда потока через расходомер нет.*)

	M0604attention: BOOL;		(*Внимание! Идет дозирование при выключенной мешалке!*)
	M0702attention: BOOL;		(*Внимание! Идет дозирование при выключенной мешалке!*)
	M0802attention: BOOL;		(*Внимание! Идет дозирование при выключенной мешалке!*)

	N0204statRegimeP1M: BOOL;		(*Статус: режим главный насос Н02.04/01.*)
	N0204statRegimeP2M: BOOL;		(*Статус: режим главный насос Н02.04/02.*)
	N0204statRegimeByC: BOOL;		(*Статус: режим Н02.04 по количеству включений.*)
	N0204statRegimeWT: BOOL;		(*Статус: режим Н02.04 по наработке.*)
	N0204workTimeP1: DWORD;		(*Счетчик времени наработки Н02.04/01.*)

	errorToOpenZD0201: BOOL;		(*Не удалось открыть ЗДЭ02.01. *)
	errorToCloseZD0201: BOOL;		(*Не удалось открыть ЗДЭ02.01*)
	errorToOpenZD0207: BOOL;		(*Не удалось открыть ЗДЭ02.07*)
	errorToCloseZD0207: BOOL;		(*Не удалось открыть ЗДЭ02.07*)
	errorToOpenZD0202: BOOL;		(*Не удалось открыть ЗДЭ02.02*)
	errorToCloseZD0202: BOOL;		(*Не удалось закрыть ЗДЭ02.02*)
	errorToOpenZD0208: BOOL;		(*Не удалось открыть ЗДЭ02.08*)
	errorToCloseZD0208: BOOL;		(*Не удалось закрыть ЗДЭ02.08*)
	errorToOpenZD0203: BOOL;		(*Не удалось открыть ЗДЭ02.03*)
	errorToCloseZD0203: BOOL;		(*Не удалось закрыть ЗДЭ02.03*)
	errorToOpenZD0209: BOOL;		(*Не удалось открыть ЗДЭ02.09*)
	errorToCloseZD0209: BOOL;		(*Не удалось открыть ЗДЭ02.09*)
	errorToOpenZD0204: BOOL;		(*Не удалось открыть ЗДЭ02.04*)
	errorToCloseZD0204: BOOL;		(*Не удалось закрыть ЗДЭ02.04*)
	errorToCloseZD0210: BOOL;		(*Не удалось закрыть ЗДЭ02.10*)
	errorToOpenZD0205: BOOL;		(*Не удалось открыть ЗДЭ02.05*)
	errorToCloseZD0205: BOOL;		(*Не удалось закрыть ЗДЭ02.05*)
	errorToOpenZD0211: BOOL;		(*Не удалось открыть ЗДЭ02.11*)
	errorToCloseZD0211: BOOL;		(*Не удалось закрыть ЗДЭ02.11*)
	regeneratedFS020106: BOOL;		(*Фильтр ФС02.01/06 промыт*)
	errorToOpenZD0206: BOOL;		(*Не удалось открыть ЗДЭ02.06*)
	errorToCloseZD0206: BOOL;		(*Не удалось закрыть ЗДЭ02.06*)
	errorToOpenZD0212: BOOL;		(*Не удалось открыть ЗДЭ02.12*)
	errorToCloseZD0212: BOOL;		(*Не удалось закрыть ЗДЭ02.12*)
	errorToOpenZD0213: BOOL;		(*Не удалось открыть ЗДЭ02.13*)
	errorToCloseZD0213: BOOL;		(*Не удалосьзакрыть ЗДЭ02.13*)
	errorToOpenZD0219: BOOL;		(*Не удалось открыть ЗДЭ02.19*)
	errorToCloseZD0219: BOOL;		(*Не удалось закрыть ЗДЭ02.19*)
	errorToOpenZD0214: BOOL;		(*Не удалось открыть ЗДЭ02.14*)
	errorToCloseZD0214: BOOL;		(*Не удалось закрыть ЗДЭ02.14*)
	errorToOpenZD0220: BOOL;		(*Не удалось открыть ЗДЭ02.20*)
	errorToCloseZD0220: BOOL;		(*Не удалось закрыть ЗДЭ02.20*)
	errorToOpenZD0215: BOOL;		(*Не удалось открыть ЗДЭ02.15*)
	errorToCloseZD0215: BOOL;		(*Не удалось закрыть ЗДЭ02.15*)
	errorToOpenZD0221: BOOL;		(*Не удалось открыть ЗДЭ02.21*)
	errorToCloseZD0221: BOOL;		(*Не удалось закрыть ЗДЭ02.21*)
	errorToOpenZD0216: BOOL;		(*Не удалось открыть ЗДЭ02.16*)
	errorToCloseZD0216: BOOL;		(*Не удалось закрыть ЗДЭ02.16*)
	errorToOpenZD0222: BOOL;		(*Не удалось открыть ЗДЭ02.22*)
	errorToCloseZD0222: BOOL;		(*Не удалось закрыть ЗДЭ02.22*)
	errorToOpenZD0217: BOOL;		(*Не удалось открыть ЗДЭ02.17*)
	errorToCloseZD0217: BOOL;		(*Не удалось закрыть ЗДЭ02.17*)
	errorToOpenZD0223: BOOL;		(*Не удалось открыть ЗДЭ02.23*)
	errorToCloseZD0223: BOOL;		(*Не удалось закрыть ЗДЭ02.23*)
	errorToOpenZD0218: BOOL;		(*Не удалось открыть ЗДЭ02.18*)
	errorToCloseZD0218: BOOL;		(*Не удалось закрыть ЗДЭ02.18*)
	errorToOpenZD0224: BOOL;		(*Не удалось открыть ЗДЭ02.24*)
	errorToCloseZD0224: BOOL;		(*Не удалось закрыть ЗДЭ02.24*)

END_VAR
VAR RETAIN
	maxTemperature: WORD;		(*Температура, выше которой будет подан сигнал ВЫСОКАЯ ТЕМПЕРАТУРА*)
	minTemperature: WORD;		(*температура, ниже которой будет подан сигнал НИЗКАЯ ТЕМПЕРАТУРА*)

	FPKtimeToWork: TIME := T#15m;		(*Задание времени на работу фильтр-пресса после спада сигнала
			уровня осадка. По умолчанию = 15мин.*)
	FPKnotStartedTime: TIME := T#3m;		(*Время задержки контроля, что ФПК запустился, после подачи на
			него сигнала на запуск. По умолчанию 3 мин.*)
	FPKmaxPressureValue: REAL := 10;		(*Максимально допустимое давление на входе ФПК. Если равно или больше,
			ФПК нужно чистить. По умолчанию = 10 (бар).*)

	FQS0301totalAmount: REAL;		(*Переменная для хранения накопленной суммы очищенных стоков от импульсного счетчика на выходе.*)

	filterTotalAmountFT0102: REAL;		(*Сумма стоков, прошедших через FT01.02.*)
END_VAR
VAR_INPUT RETAIN
	ND0502setMaxDosVal: REAL;		(*Указать максимальную производительность НД05.02.*)
	ND0502setKoefProp: REAL := 126.39;		(*Задать количество реагента в мл на один кубометр стоков.
			По умолчанию = 126,39.*)
	ND0502regimeP1M: BOOL;		(*Выбор режима включения доз.насосов НД05.02: первый насос - главный.
			*)
	ND0502regimeP2M: BOOL;		(*Выбор режима включения доз.насосов НД05.02:
			второй насос - главный.*)
	ND0502regimeByWT: BOOL;		(*Выбор режима включения доз.насосов НД05.02:
			по наработке.*)
	ND0502regimeByC: BOOL;		(*Выбор режима включения доз.насосов НД05.02:
			по количеству включений.*)

	ND0602setMaxDosVal: REAL;		(*Указать максимальную производительность НД06.02.*)
	ND0602setKoefProp: REAL := 145.83;		(*Задать количество реагента в мл на один кубометр стоков.
			По умолчанию - 145,83.*)
	ND0602regimeP1M: BOOL;		(*Выбор режима включения доз.насосов НД06.02: первый насос - главный.
			*)
	ND0602regimeP2M: BOOL;		(*Выбор режима включения доз.насосов НД06.02: второй насос - главный.
			*)
	ND0602regimeByWT: BOOL;		(*Выбор режима включения доз.насосов НД06.02:
			по наработке.*)
	ND0602regimeByC: BOOL;		(*Выбор режима включения доз.насосов НД06.02:
			по количеству включений.*)

	ND0603setMaxDosVal: REAL;		(*Указать максимальную производительность НД06.03.*)
	ND0603setKoefProp: REAL := 145.83;		(*Задать количество реагента в мл на один кубометр стоков.
			По умолчанию = 145,83.*)
	ND0603regimeP1M: BOOL;		(*Выбор режима включения доз.насосов НД06.03: первый насос - главный.
			*)
	ND0603regimeP2M: BOOL;		(*Выбор режима включения доз.насосов НД06.03: второй насос - главный.*)
	ND0603regimeByWT: BOOL;		(*Выбор режима включения доз.насосов НД06.03:
			по наработке.*)
	ND0603regimeByC: BOOL;		(*Выбор режима включения доз.насосов НД06.03:
			по количеству включений.*)

	ND0703pHsetValue: REAL := 7.5;		(*Задание рН для поддержания подачей щелочи НД07.03 и контроля по QE01.01.*)
	ND0703regimeP1M: BOOL;		(*Выбор режима включения доз.насосов НД07.03: первый насос - главный.
			*)
	ND0703regimeP2M: BOOL;		(*Выбор режима включения доз.насосов НД07.03: второй насос - главный*)
	ND0703regimeByWT: BOOL;		(*Выбор режима включения доз.насосов НД07.03: по наработке.*)
	ND0703regimeByC: BOOL;		(*Выбор режима включения доз.насосов НД07.03: по количеству включений.*)
	ND0703koeffI: REAL := 10;		(*Коэффициент интегральной части ПИД. По умолчанию = 10.*)
	ND0703koeffD: REAL := 1;		(*Коэффициент дифференциальной части ПИД. По умолчанию = 1.*)
	ND0703koeffP: REAL := 1;		(*Коэффициент пропорциональной части ПИД. По умолчанию = 1.*)

	ND0803setMaxDosVal: REAL;		(*Указать максимальную производительность НД08.03*)
	ND0803setKoefProp: REAL := 576.53;		(*Задать количество реагента в мл на один кубометр стоков.
			По умолчанию = 576,53.*)
	ND0803regimeP1M: BOOL;		(*Выбор режима включения доз.насосов НД08.03: первый насос - главный.
			*)
	ND0803regimeP2M: BOOL;		(*Выбор режима включения доз.насосов НД08.03: второй насос - главный.*)
	ND0803regimeByWT: BOOL;		(*Выбор режима включения доз.насосов НД08.03: по наработке.*)
	ND0803regimeByC: BOOL;		(*Выбор режима включения доз.насосов НД08.03: по количеству включений.*)

	ND0804doseValue: WORD := 100;		(*Задание на дозирование НД0804 в процентах от максимальной
			производительности (0-100%). По умолчанию = 100.*)

	N0105regimeByC: BOOL;		(*Выбор режима запуска Н01.05: по количеству включений.	*)
	N0105regimeByWT: BOOL;		(*Выбор режима запуска Н01.05: по наработке.*)
	N0105flowSetValue: REAL := 72;		(*Задание расхода для поддержания ЧРП Н01.05 по расходомеру FT01.02.
			По умолчанию = 72 кубометра в час.*)
	N0105koeffP: REAL := 1;		(*Коэффициент пропорциональной части ПИД. По умолчанию = 1.*)
	N0105koeffI: REAL := 10;		(*Коэффициент интегральной части ПИД. По умолчанию = 10.*)
	N0105koeffD: REAL := 1;		(*Коэффициент дифференциальной части ПИД. По умолчанию = 1.*)
	N0105minFlowTime: TIME := T#60s;		(*Время на создание потока включенным насосом.
			По умолчанию = 60сек. Если не создал = авария.*)

	timeToOpenCloseValve: TIME := T#30s;		(*Время на открытие/закрытие заслонки. Общее для всех заслонок.
			По умолчанию равно 30 секунд.*)

	N0404regimeP1M: BOOL;		(*Выбор режима с главным насосом Н04.04/01.*)
	N0404regimeP2M: BOOL;		(*Выбор режима с главным насосом Н04.04/02.*)
	N0404regimeByC: BOOL;		(*Выбор режима, запуск по количеству включений.*)
	N0404regimeWT: BOOL;		(*Выбор режима, по наработке.*)

	UFO0301startDelayTime: TIME := T#3m;		(*Время задержки запуска УФО после начала протекания стоков.
			По умолчанию = 3мин.*)
	UFO0301regimeP1M: BOOL;		(*Выбор режима главное УФО: 03.01/01.*)
	UFO0301regimeP2M: BOOL;		(*Выбор режима главное УФО: 03.01/02.*)
	UFO0301regimeByC: BOOL;		(*Выбор режима УФО по количеству включений (выбирается по умолчанию).*)
	UFO0301regimeWT: BOOL;		(*Выбор режима УФО по наработке.*)

	FQS0301impulsValue: REAL := 0.1;		(*Вес импульса расходомера.
			По умолчанию = 0,1 кубометр.*)

	N0204regimeP1M: BOOL;		(*Выбор режима главный: Н02.04/01*)
	N0204regimeP2M: BOOL;		(*Выбор режима главный: Н02.04/02*)
	N0204regimeByC: BOOL;		(*Выбор режима Н02.04 по количеству включений (по умолчанию).*)
	N0204regimeWT: BOOL;		(*Выбор режима Н02.04 по наработке.*)

	filterValueToRegen: REAL := 1000;		(*Величина объема стоков для отправки фильтра на промывку (регенерацию).
			По умолчанию = 1000.*)

END_VAR
VAR_OUTPUT RETAIN
	ND0502counterP1: WORD;		(*Счетчик количества включений НД05.02/01.*)
	ND0502counterP2: WORD;		(*Счетчик количества включений НД05.02/02.*)
	ND0502workTimeP1: DWORD;		(*Счетчик времени наработки НД05.02/01.*)
	ND0502workTimeP2: DWORD;		(*Счетчик времени наработки НД05.02/02.*)

	ND0602counterP1: WORD;		(*Счетчик количества включений НД06.02/01.*)
	ND0602counterP2: WORD;		(*Счетчик количества включений НД06.02/02.*)
	ND0602workTimeP1: DWORD;		(*Счетчик времени наработки НД06.02/01.*)
	ND0602workTimeP2: DWORD;		(*Счетчик времени наработки НД06.02/02.*)

	ND0603counterP1: WORD;		(*Счетчик количества включений НД06.03/01.*)
	ND0603counterP2: WORD;		(*Счетчик количества включений НД06.03/02.*)
	ND0603workTimeP1: DWORD;		(*Счетчик времени наработки НД06.03/01.*)
	ND0603workTimeP2: DWORD;		(*Счетчик времени наработки НД06.03/02.*)

	ND0703counterP1: WORD;		(*Счетчик количества включений НД07.03/01.*)
	ND0703counterP2: WORD;		(*Счетчик количества включений НД07.03/02.*)
	ND0703workTimeP1: DWORD;		(*Счетчик времени наработки НД07.03/01.*)
	ND0703workTimeP2: DWORD;		(*Счетчик времени наработки НД07.03/02.*)

	ND0803counterP1: WORD;		(*Счетчик количества включений НД08.03/01.*)
	ND0803counterP2: WORD;		(*Счетчик количества включений НД08.03/02.*)
	ND0803workTimeP1: DWORD;		(*Счетчик времени наработки НД08.03/01.*)
	ND0803workTimeP2: DWORD;		(*Счетчик времени наработки НД08.03/02.*)

	N0105counterP1: WORD;		(*Счетчик количества включений Н01.05/01.*)
	N0105counterP2: WORD;		(*Счетчик количества включений Н01.05/02.*)
	N0105workTimeP1: DWORD;		(*Счетчик времени наработки Н01.05/01.*)
	N0105workTimeP2: DWORD;		(*Счетчик времени наработки Н01.05/02.*)

	N0404counterP1: WORD;		(*Счетчик количества включений Н04.04/01.*)
	N0404counterP2: WORD;		(*Счетчик количества включений Н04.04/02.*)
	N0404workTimeP1: DWORD;		(*Счетчик времени наработки Н04.04/01.*)
	N0404workTimeP2: DWORD;		(*Счетчик времени наработки Н04.04/02.*)

	UFO0301counterP1: WORD;		(*Счетчик количества включений УФО: 03.01/01.*)
	UFO0301counterP2: WORD;		(*Счетчик количества включений УФО: 03.01/02.*)
	UFO0301workTimeP1: DWORD;		(*Счетчик времени наработки УФО: 03.01/01.*)
	UFO0301workTimeP2: DWORD;		(*Счетчик времени наработки УФО: 03.01/02.*)

	FQS0301totalAmountUDINT: UDINT;		(*Общий объем стоков в целочисленном виде.*)

	N0204counterP1: WORD;		(*Счетчик количества включений Н02.04/01.*)
	N0204counterP2: WORD;		(*Счетчик количества включений Н02.04/02.*)
	N0204workTimeP2: DWORD;		(*Счетчик времени наработки Н02.04/02.*)

END_VAR
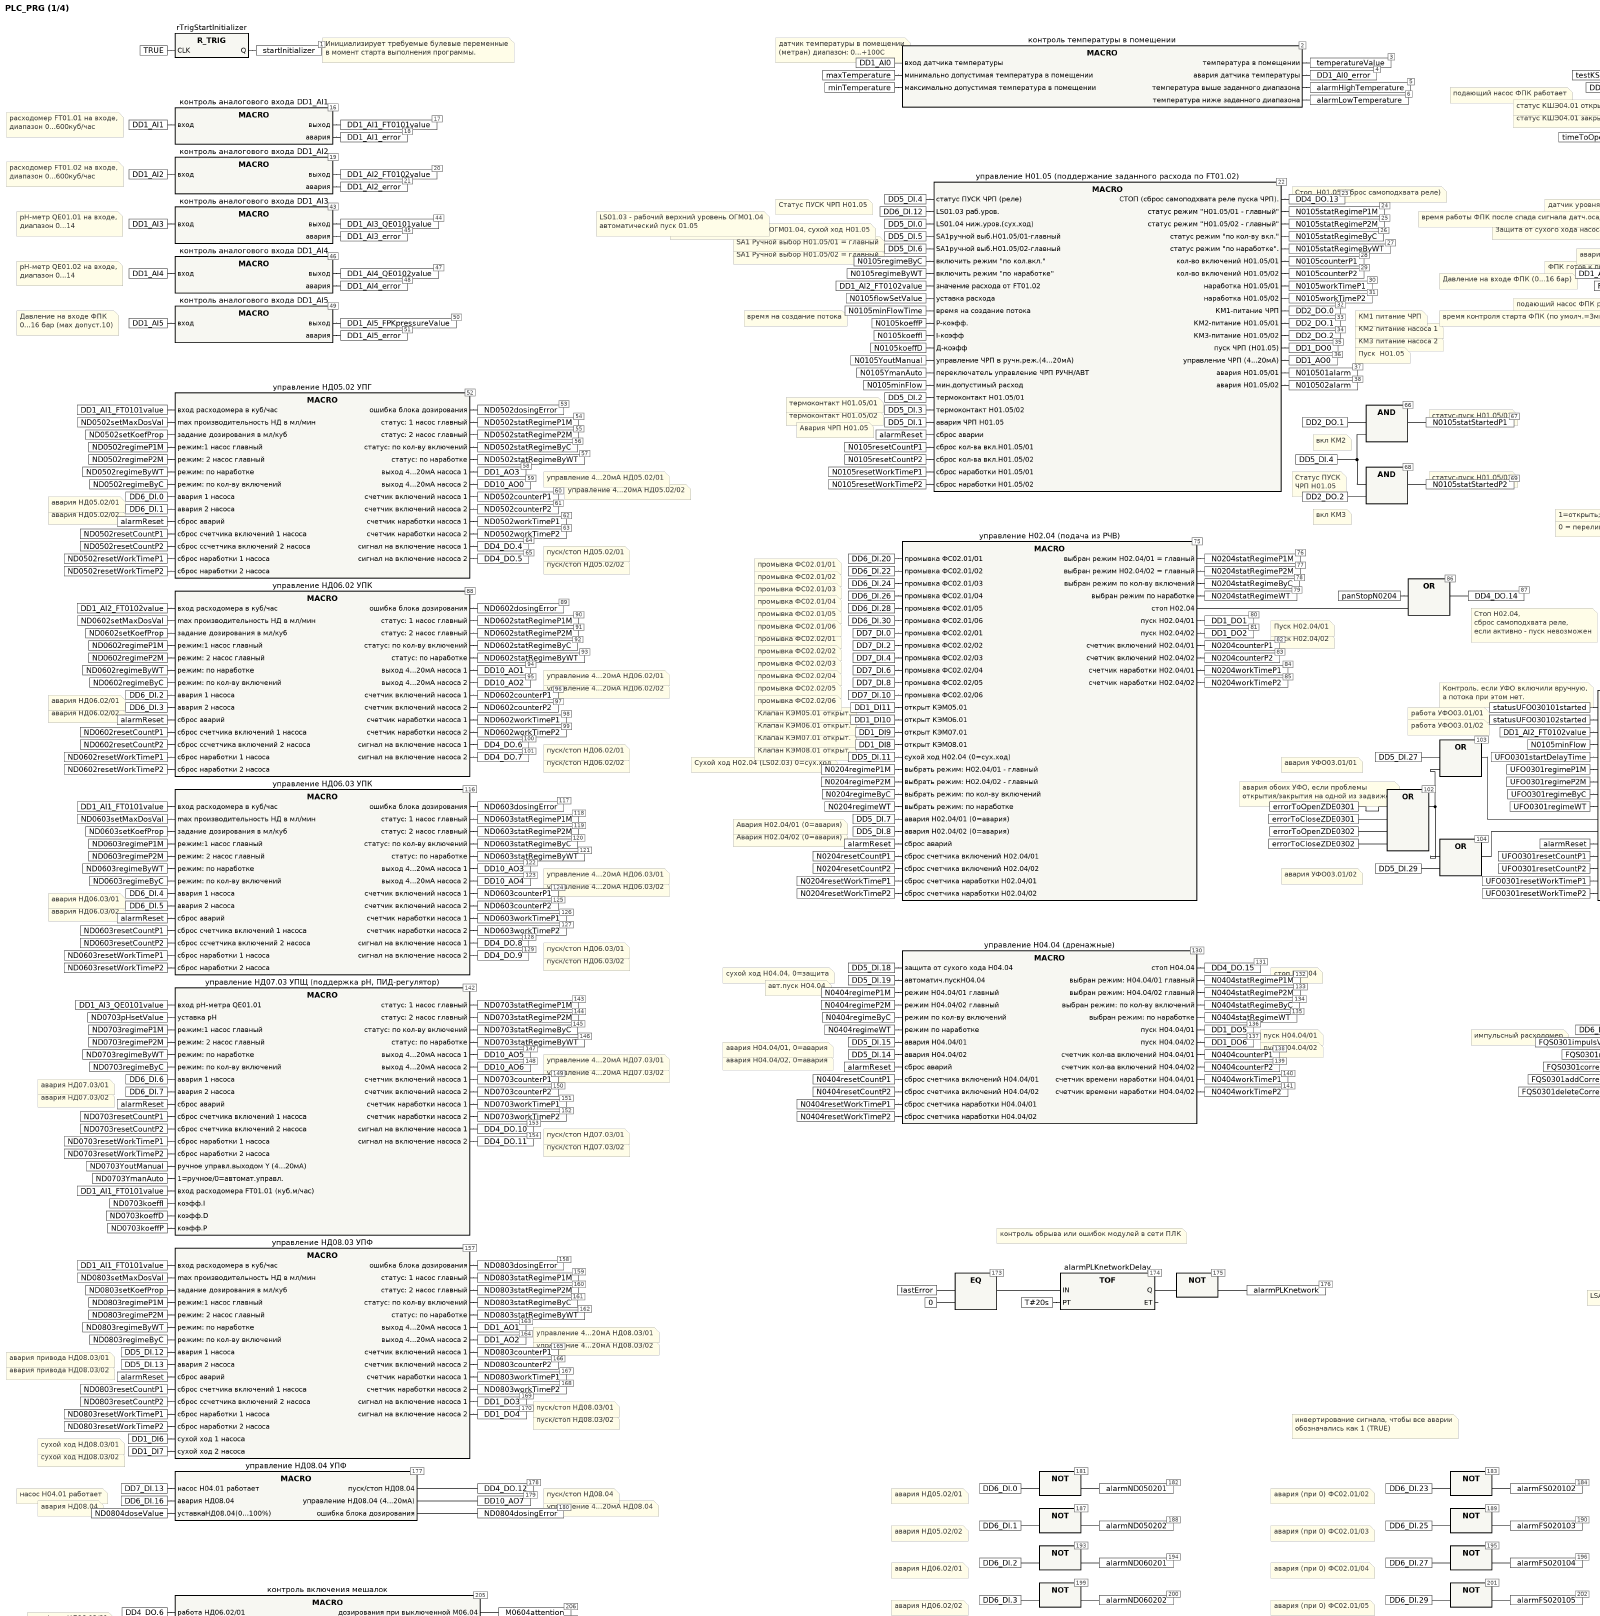
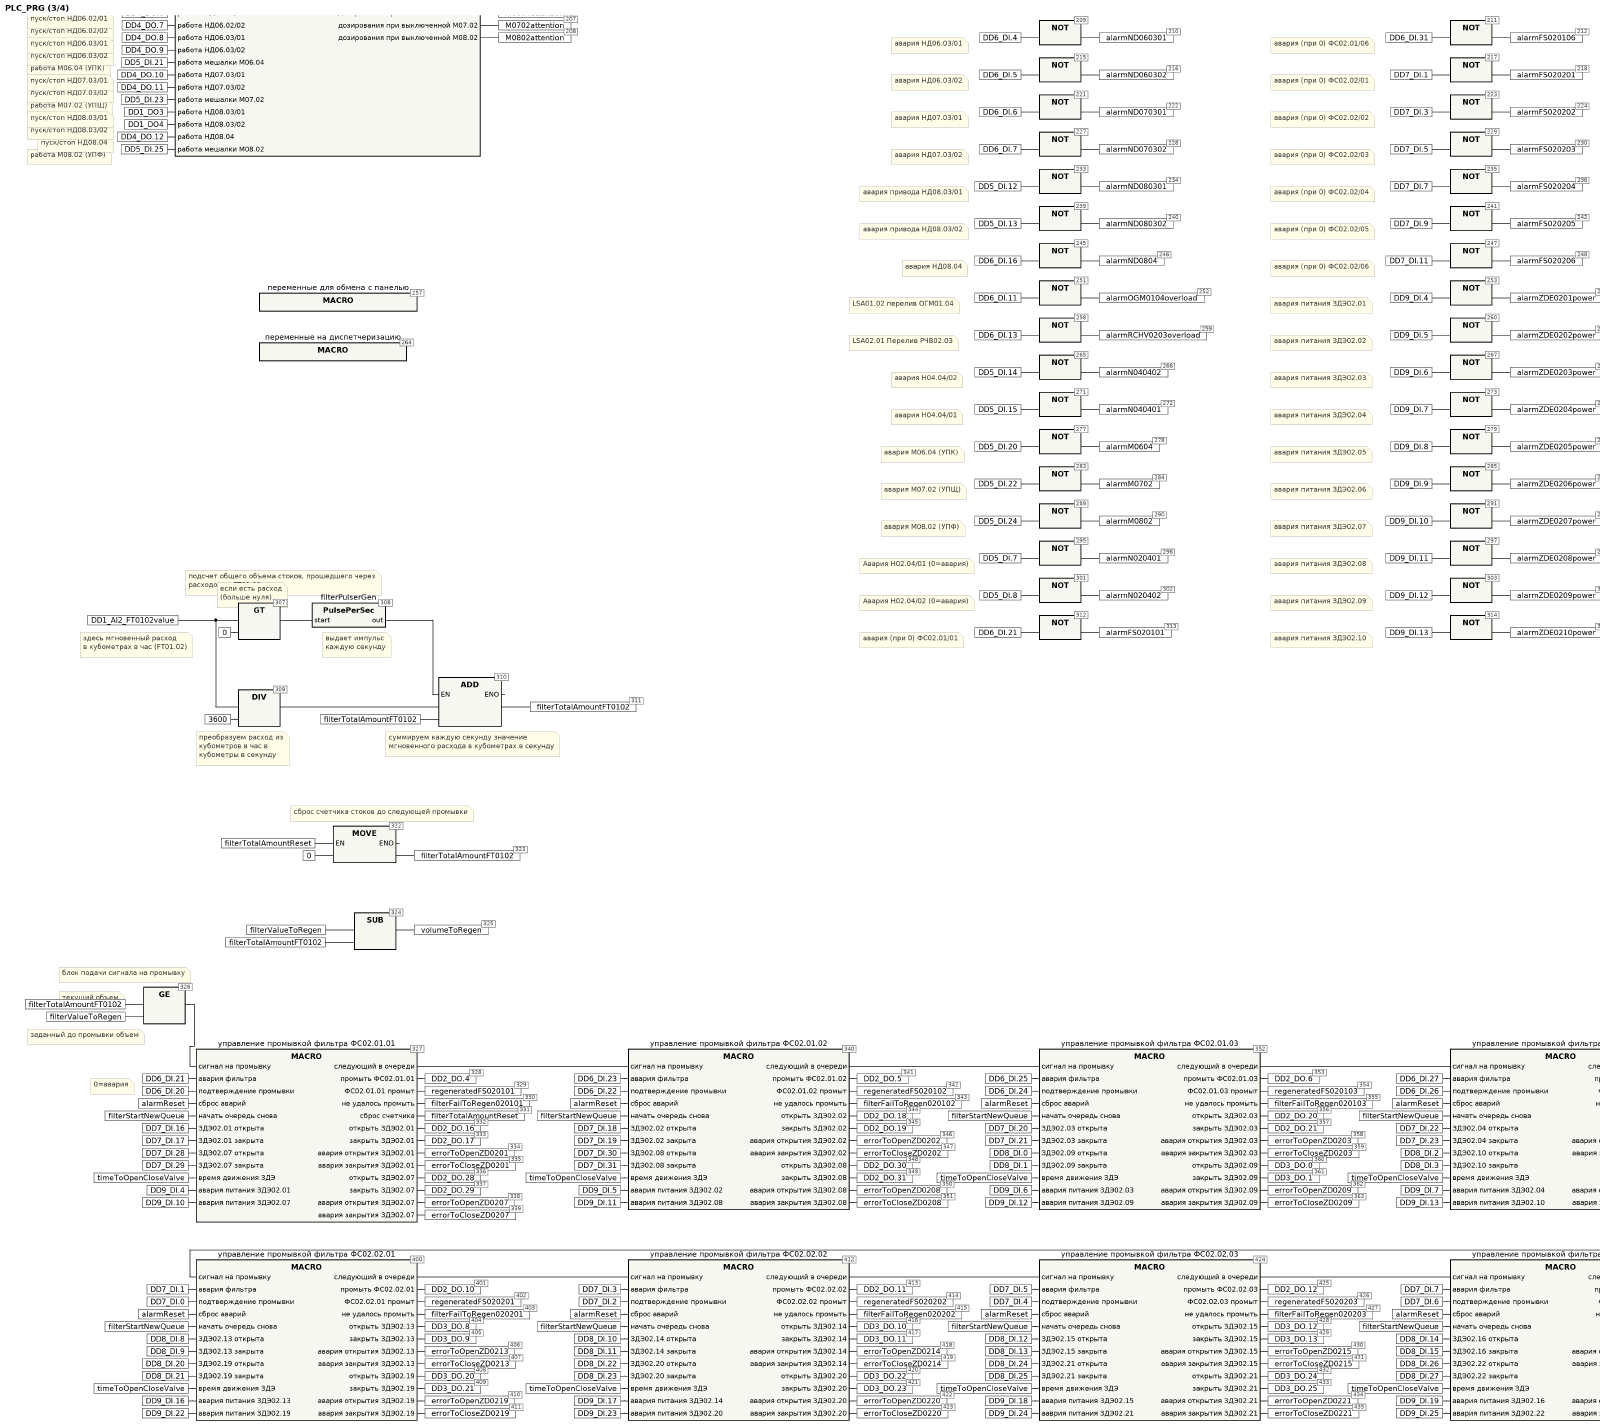
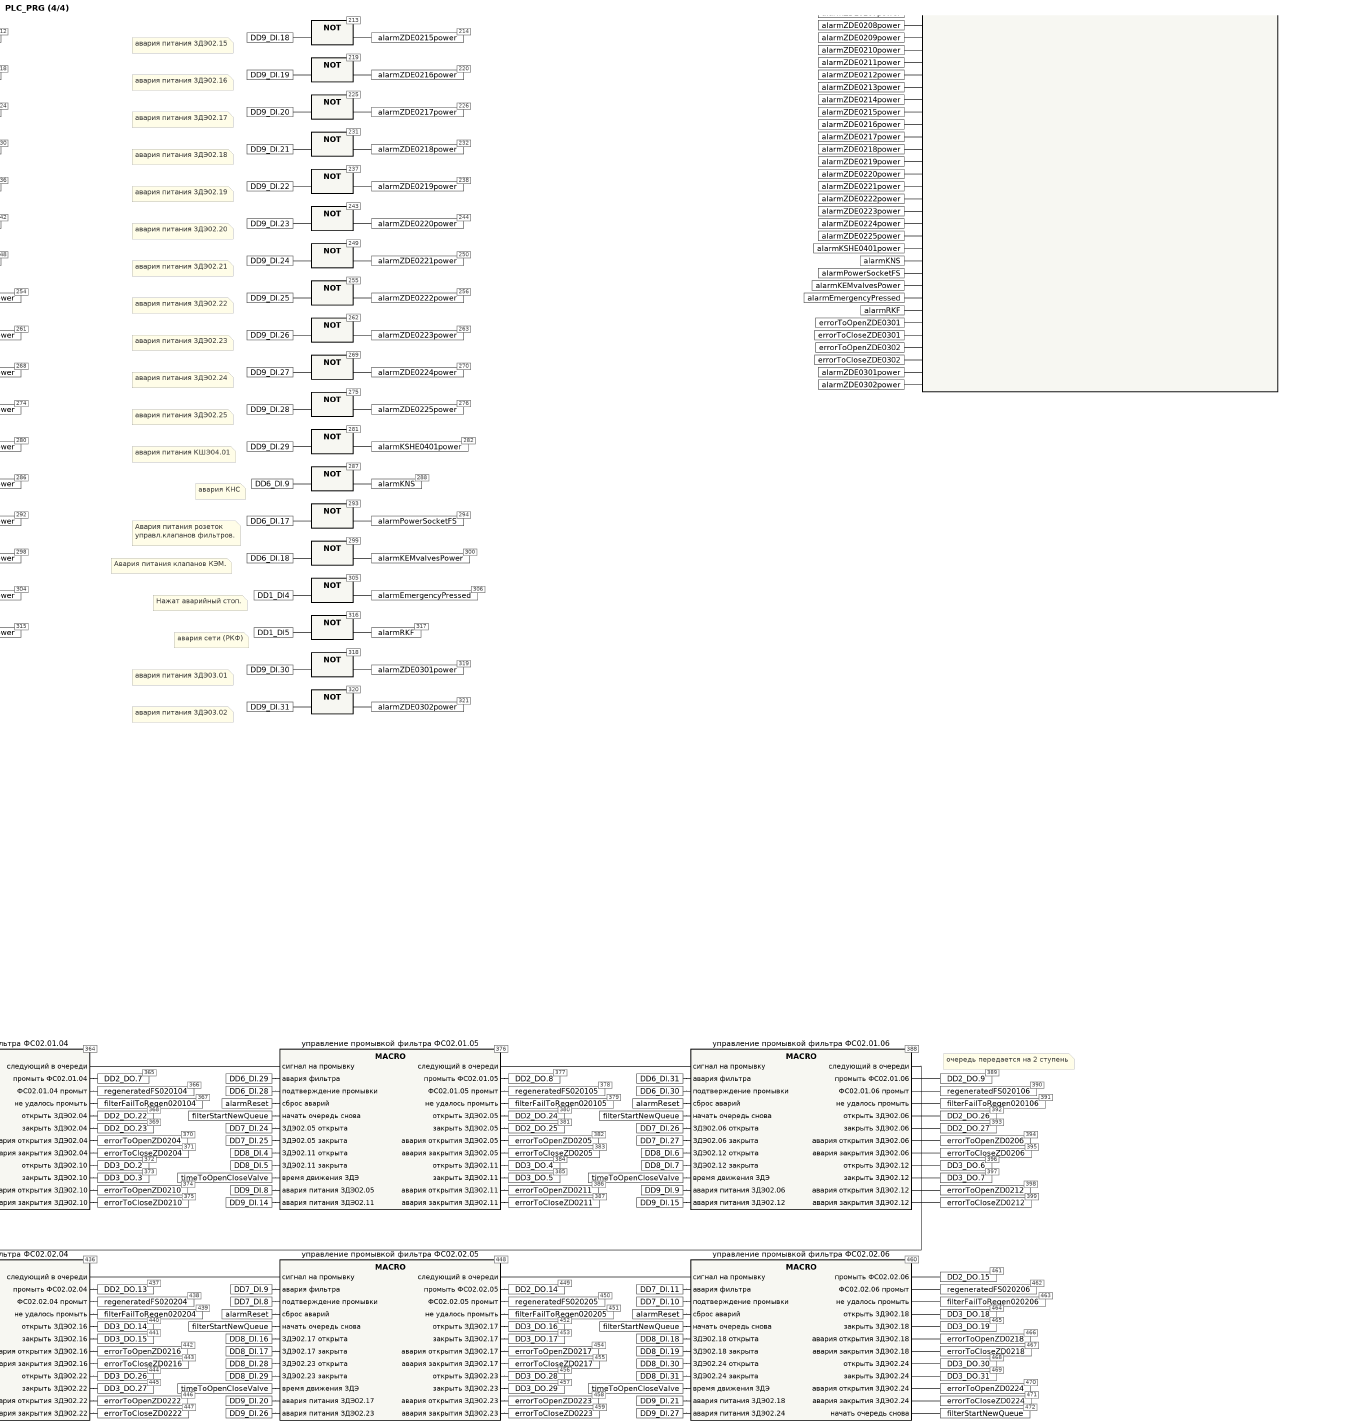
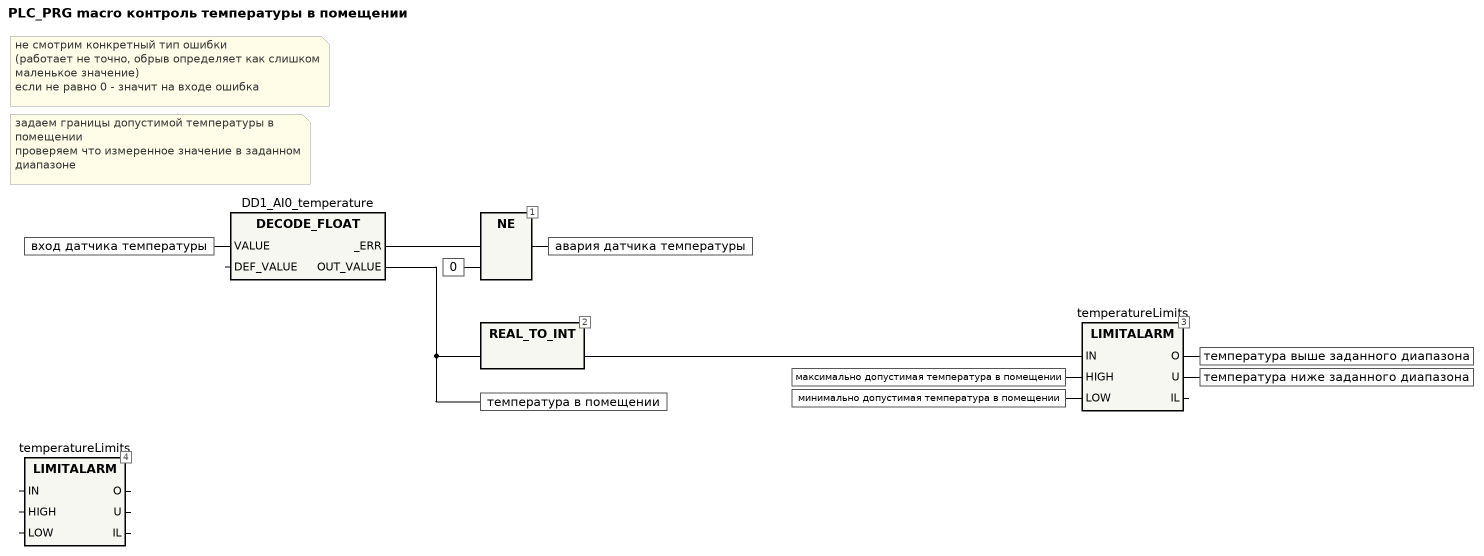
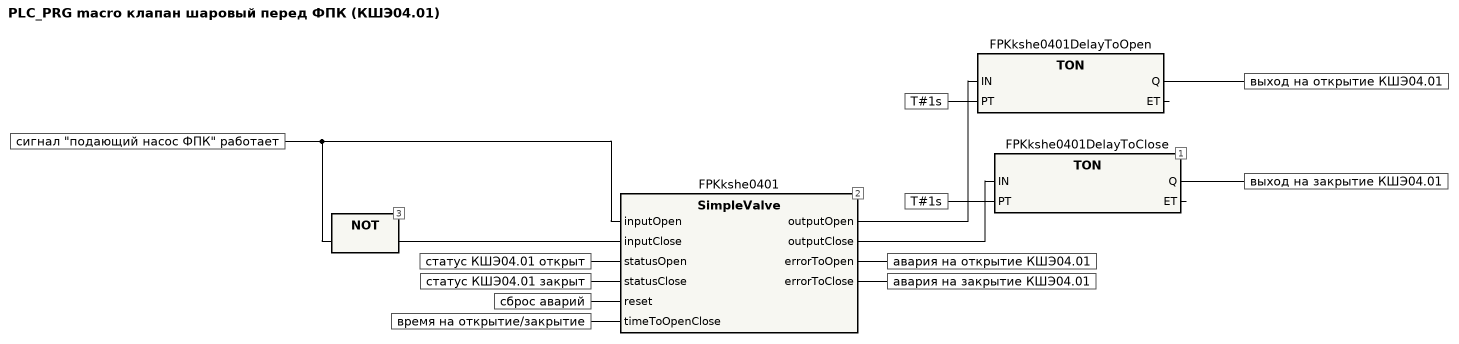
[picture p5: PLC_PRG macro клапан шаровый перед ФПК (КШЭ04.01) (CFC)]
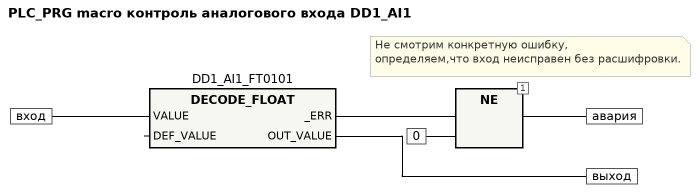
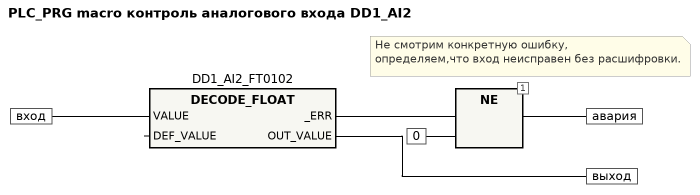
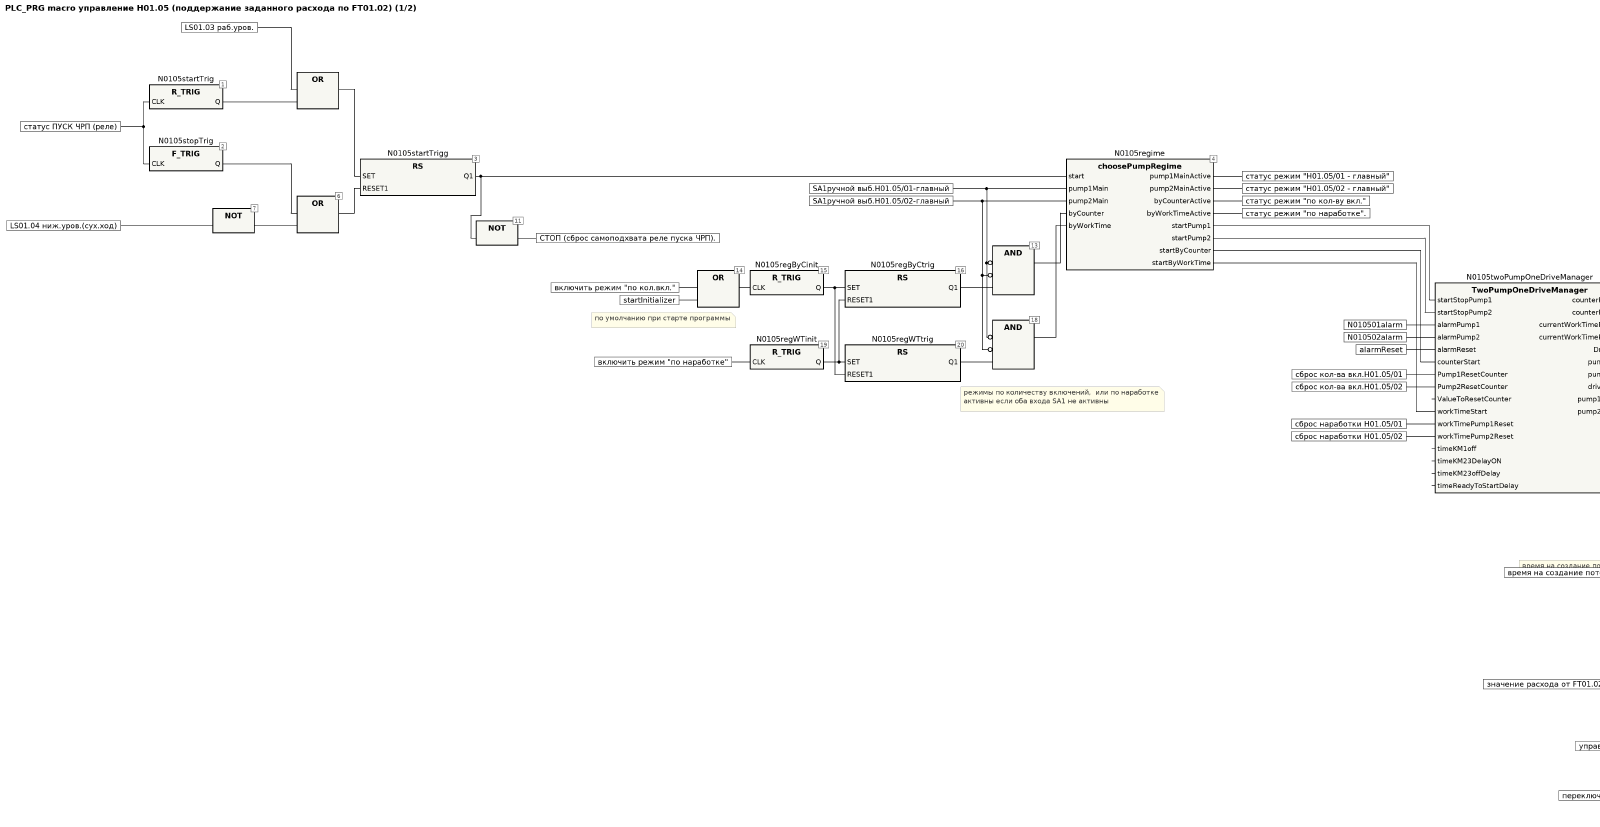
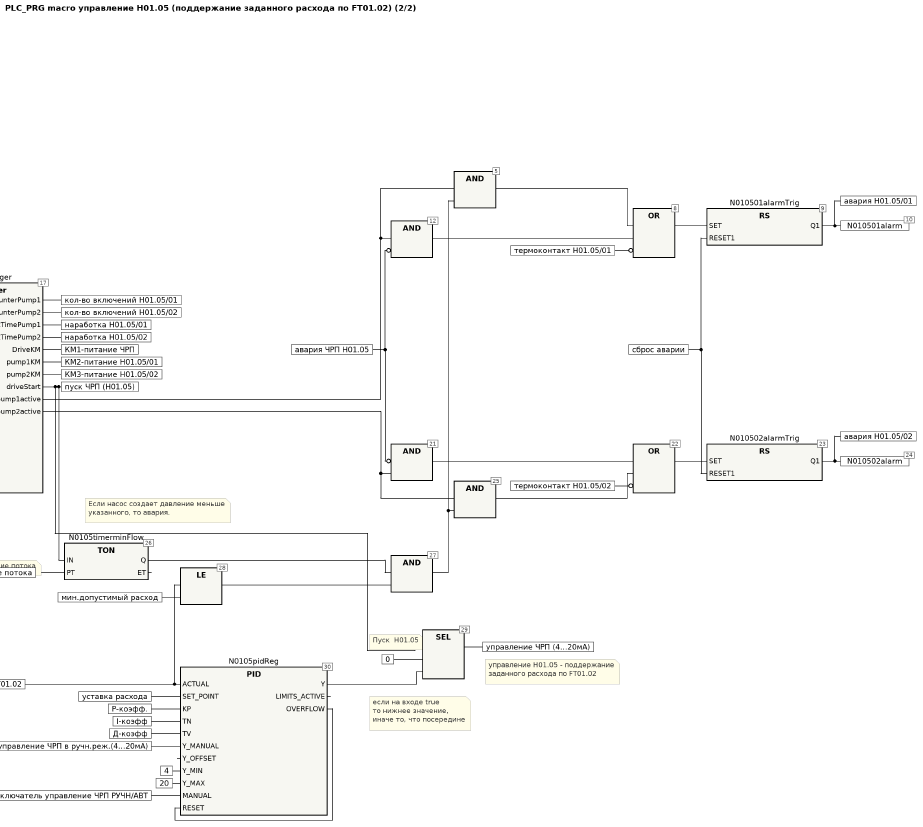
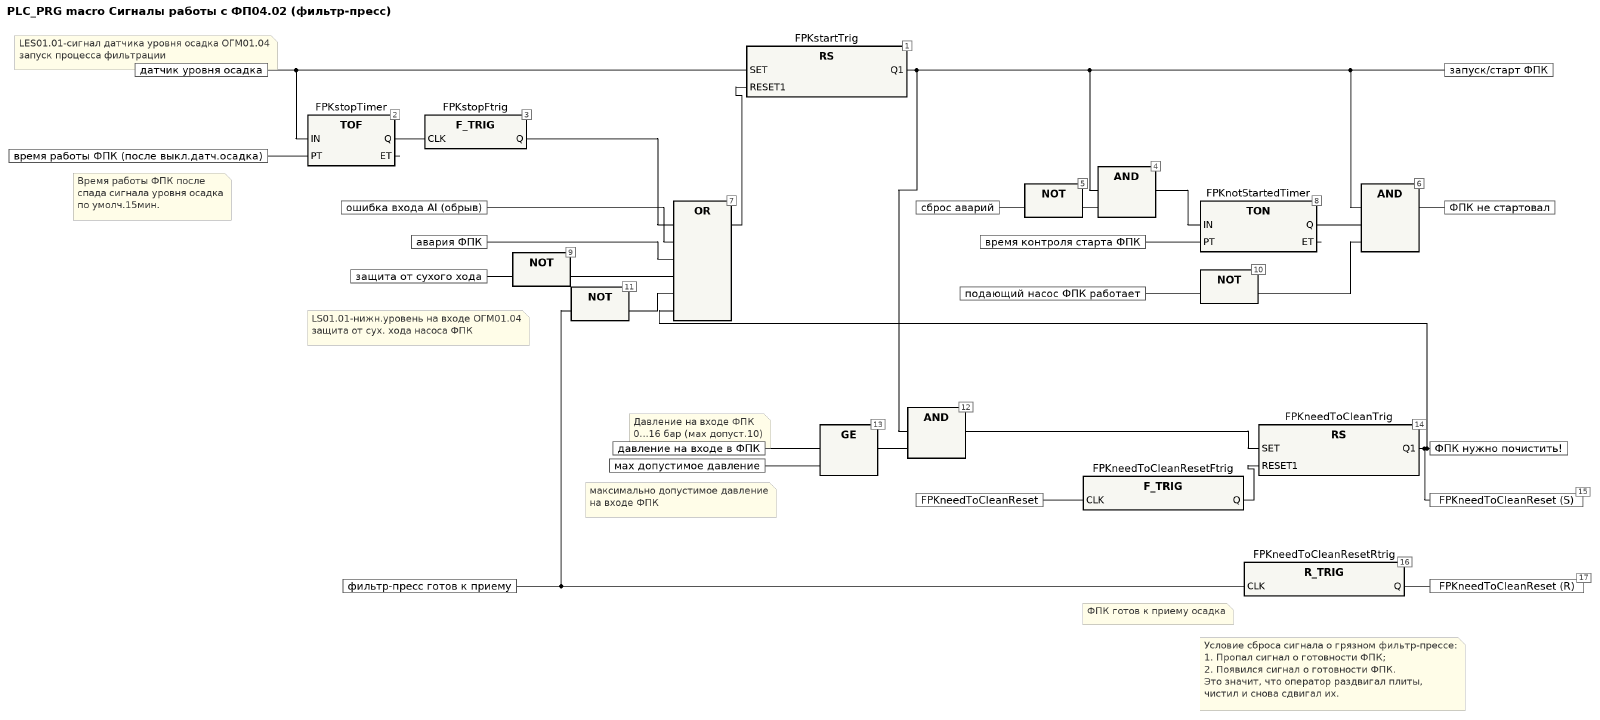
[picture p10: PLC_PRG macro Сигналы работы с ФП04.02 (фильтр-пресс) (CFC)]
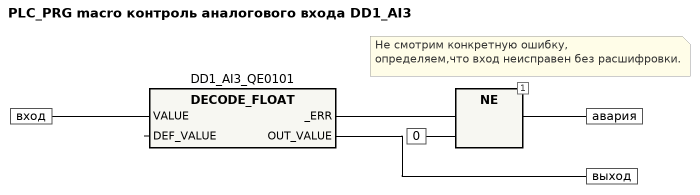
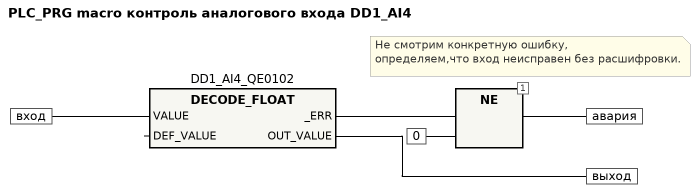
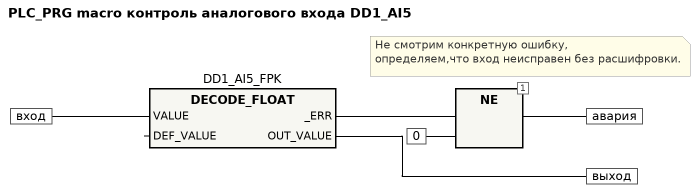
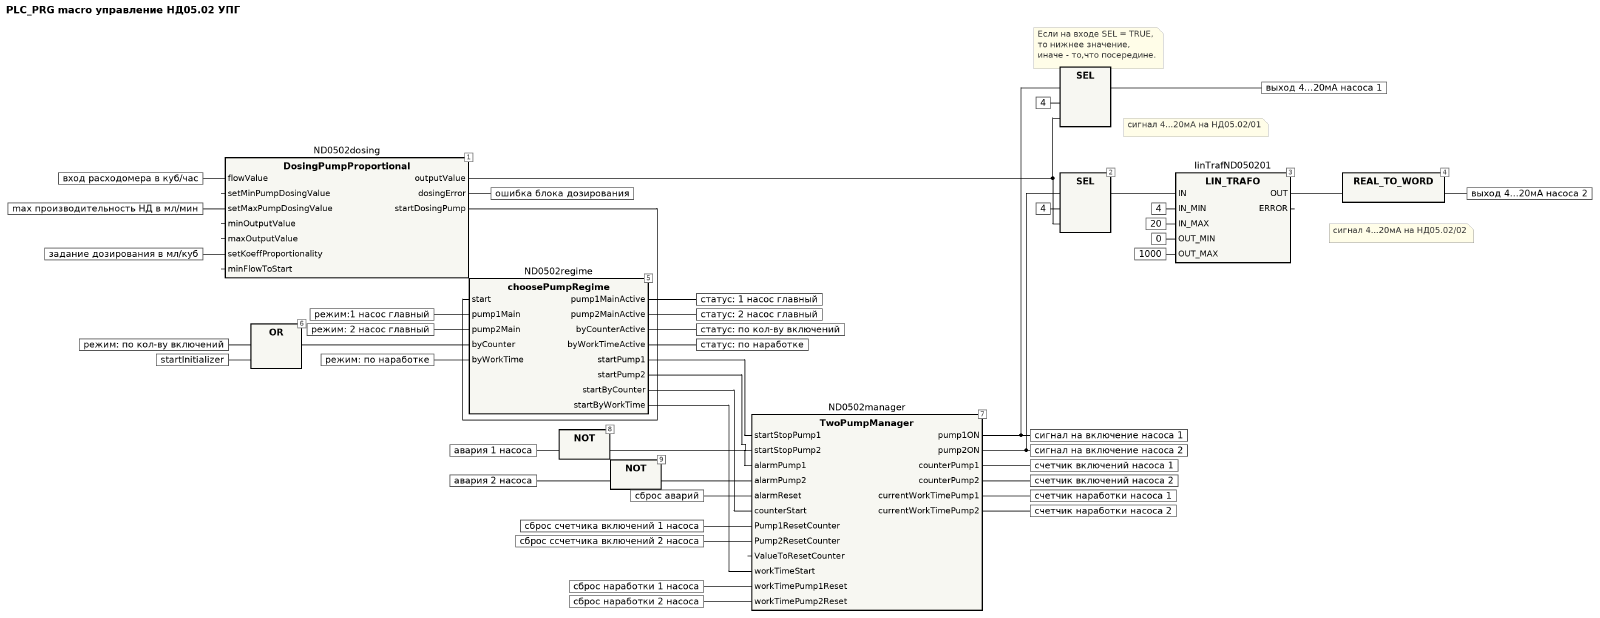
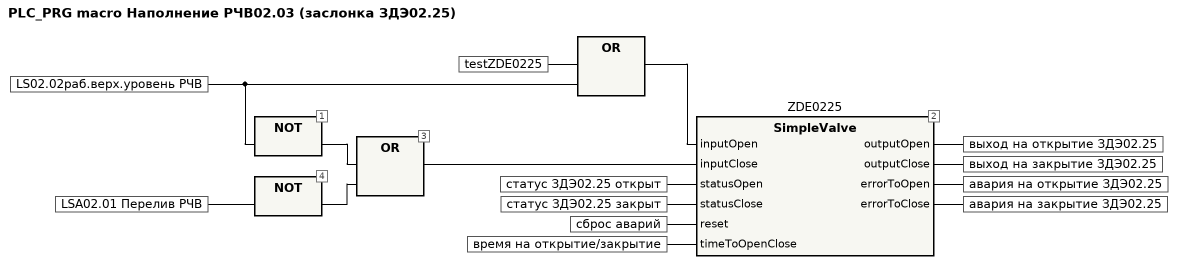
[picture p15: PLC_PRG macro Наполнение РЧВ02.03 (заслонка ЗДЭ02.25) (CFC)]
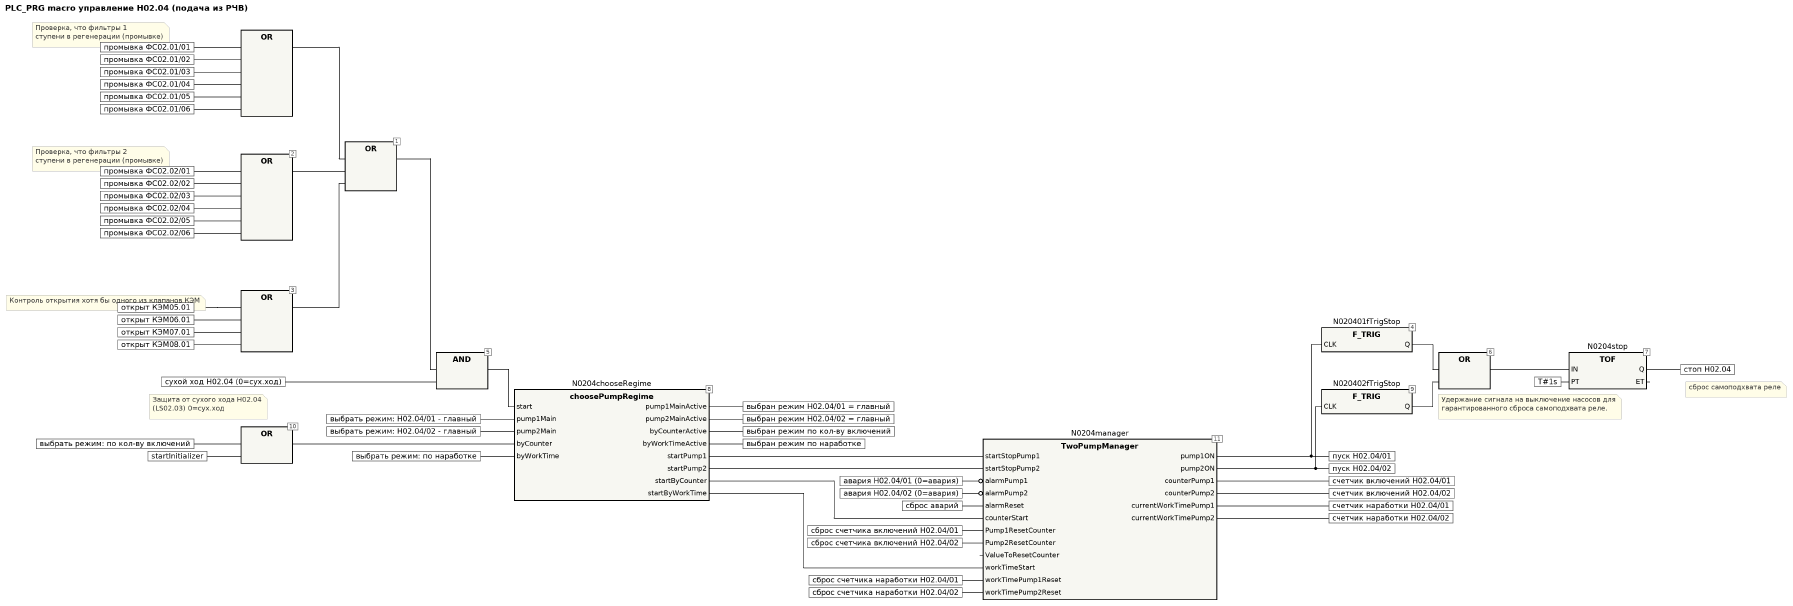
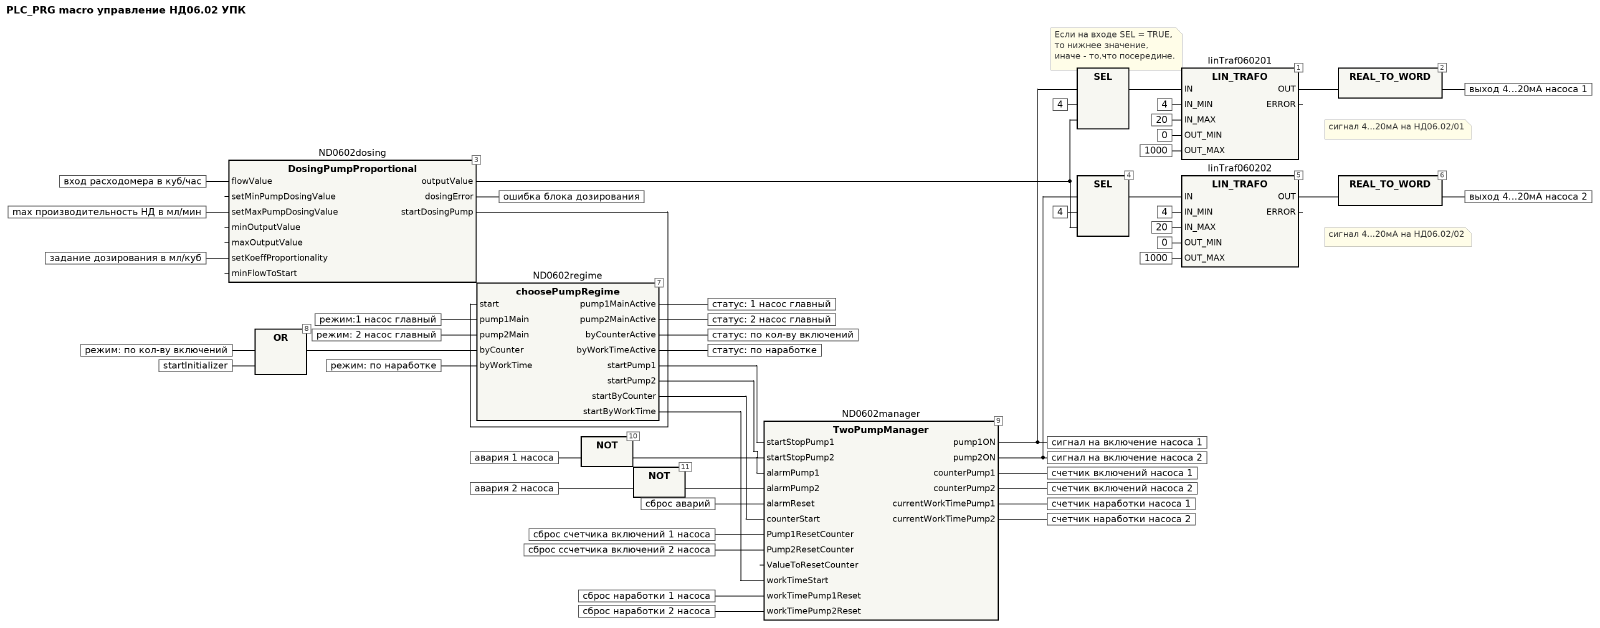
[picture p17: PLC_PRG macro управление НД06.02 УПК (CFC)]
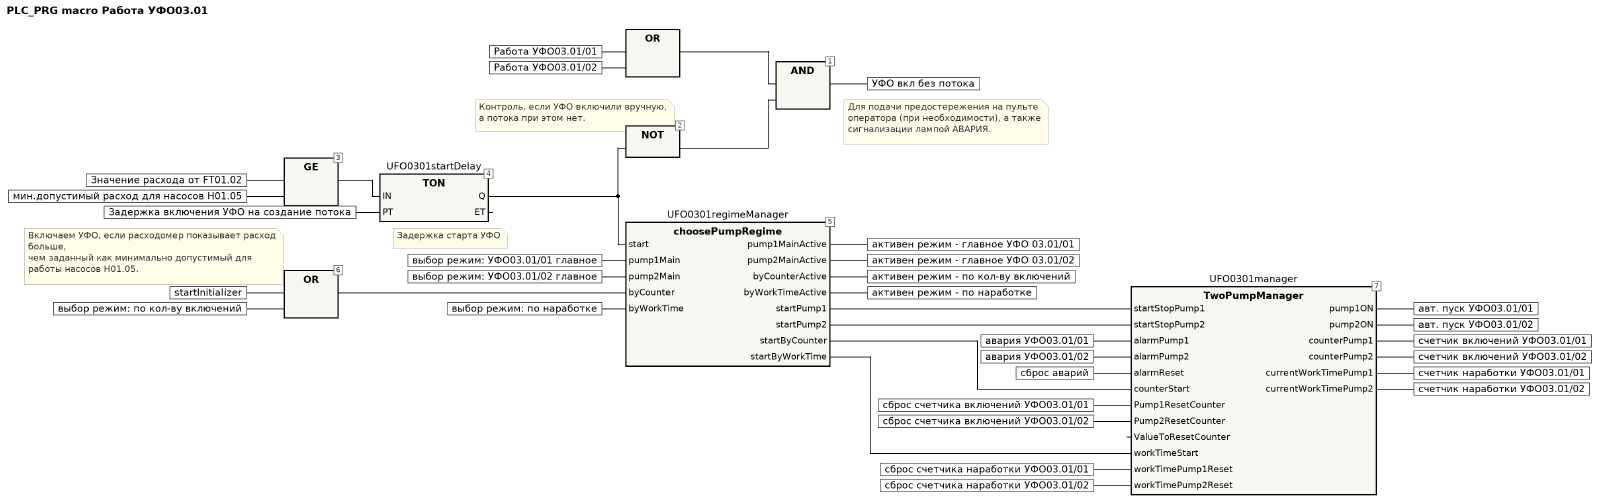
[picture p18: PLC_PRG macro Работа УФО03.01 (CFC)]
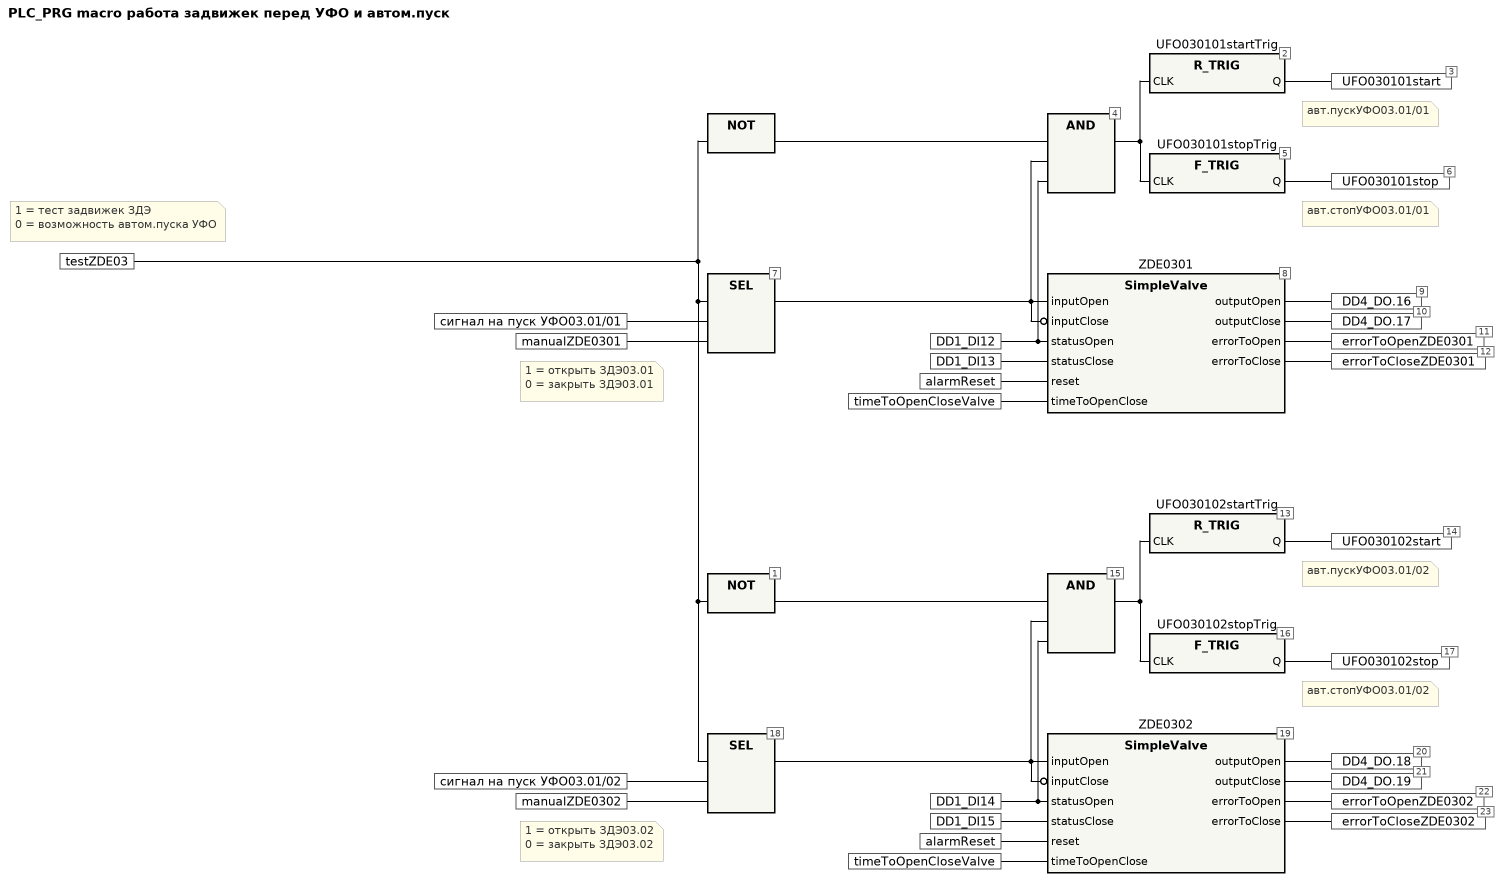
[picture p19: PLC_PRG macro работа задвижек перед УФО и автом.пуск (CFC)]
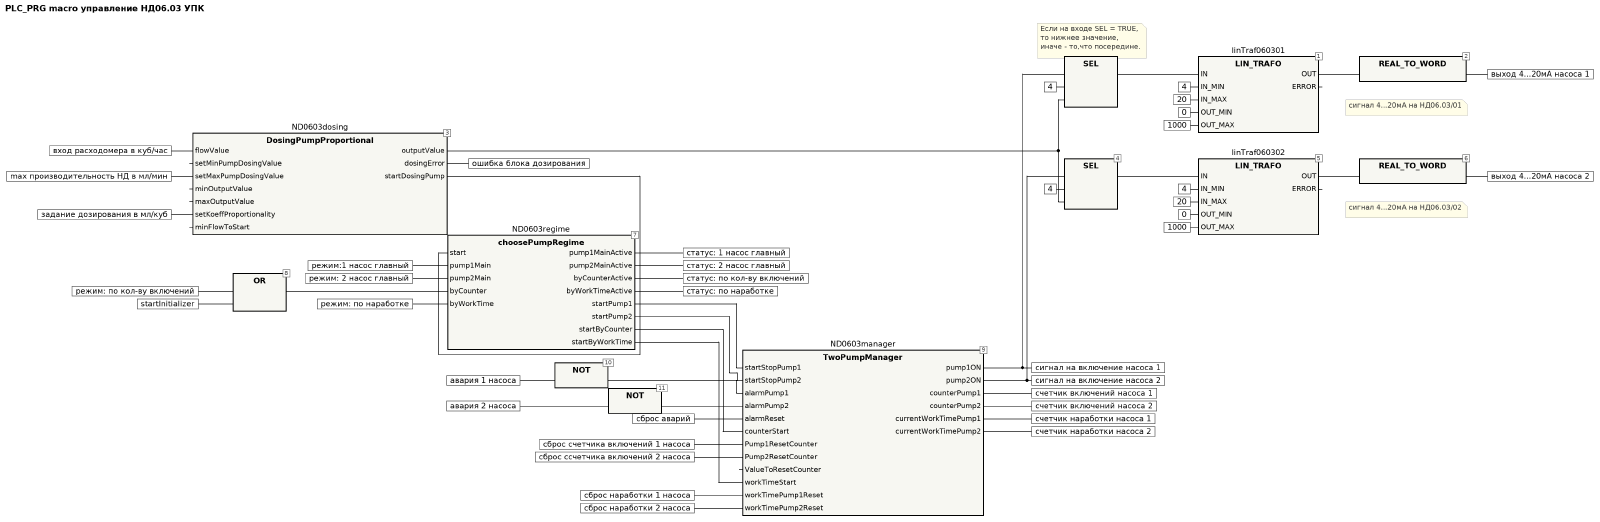
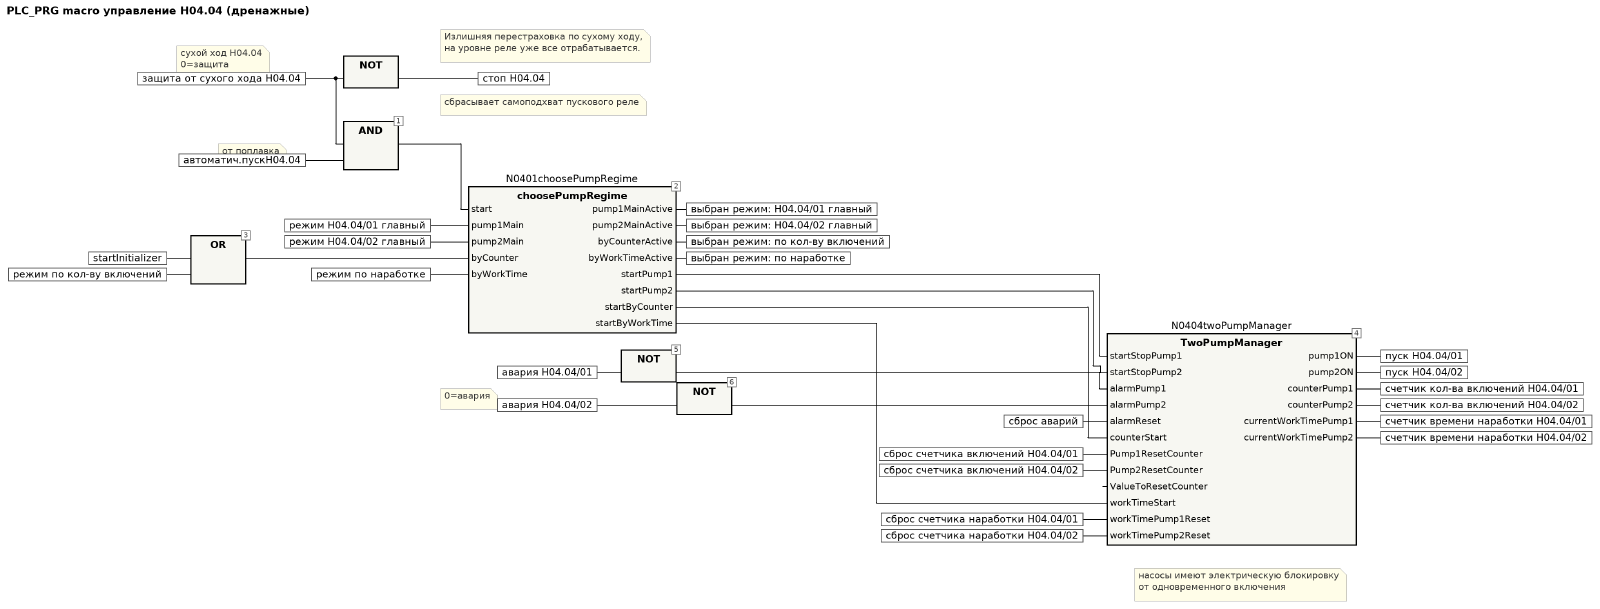
[picture p21: PLC_PRG macro управление Н04.04 (дренажные) (CFC)]
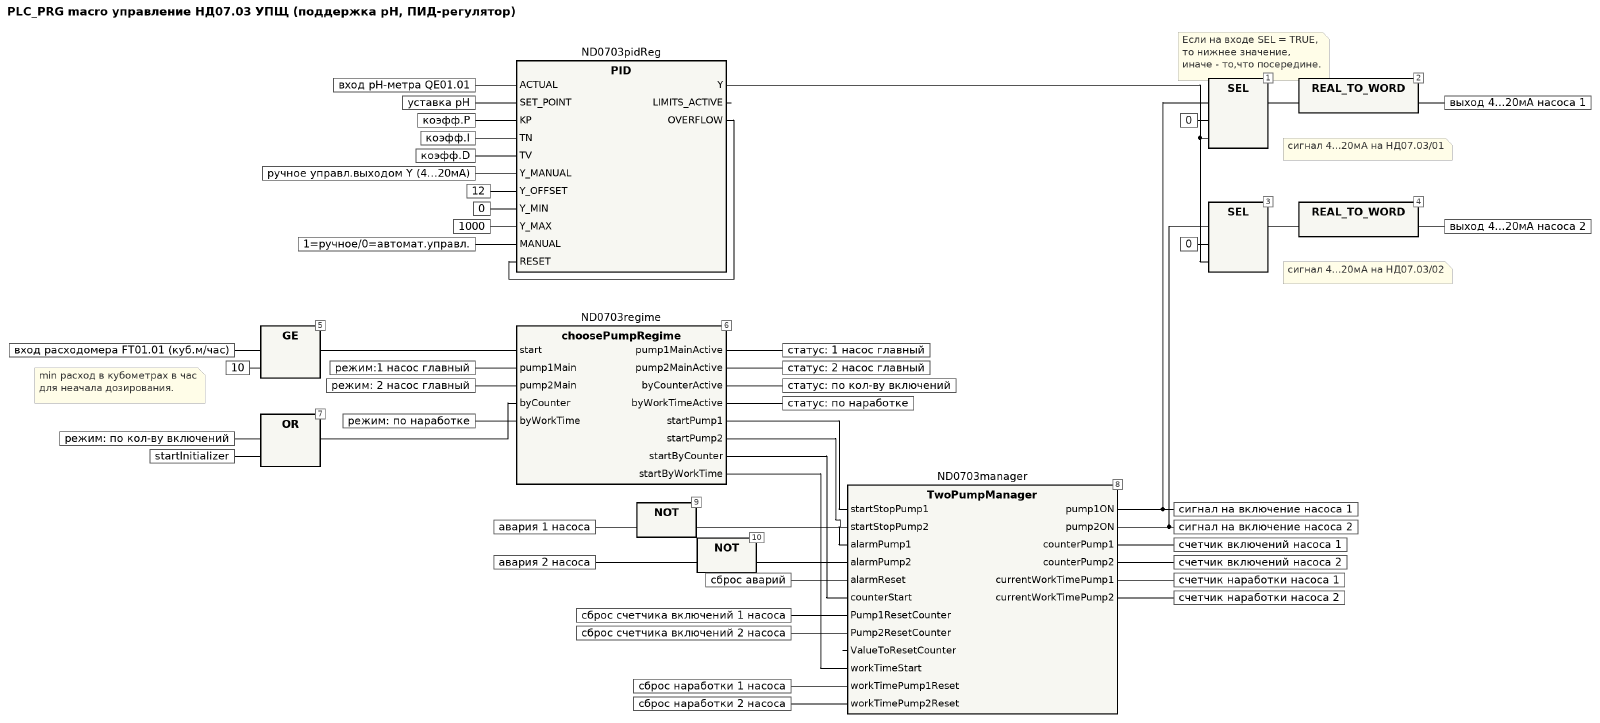
[picture p22: PLC_PRG macro управление НД07.03 УПЩ (поддержка рН, ПИД-регулятор) (CFC)]
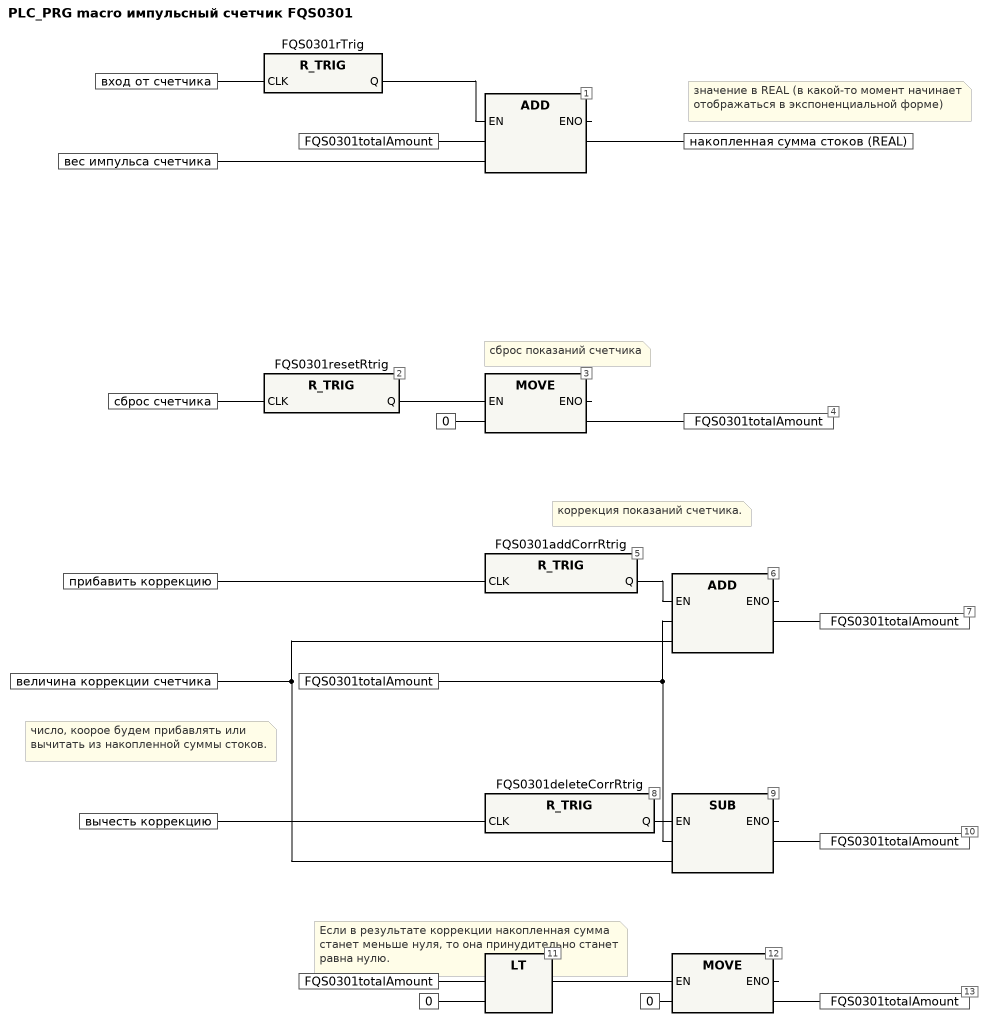
[picture p23: PLC_PRG macro импульсный счетчик FQS0301 (CFC)]
